	FOR z:=1 TO 100 DO
		IF  eRFID[z].nCardNumber=eLidFeederPackageState[2].nCardNumber AND eLidFeederPackageState[2].nCardNumber >0 THEN
			eRFID[z]:=eLidFeederPackageState[2];
		EXIT;
		END_IF;
	END_FOR 
			 
END_IF
END_ACTION

ACTION aP07_CapPusher:
	IF bCapPusherEnable THEN
	
	// SZLABAN **************************************************************************************************
	P07_CapPusher.IbCapPusherFormSensor;
	P07_CapPusher.bReadedCard;
	
	fbIbCapPusherFormSensor	(bIn:=	P07_CapPusher.IbCapPusherFormSensor AND 
									P07_CapPusher.bReadedCard AND
									fbPMLAuto.ePMLState = Tc3_PackML.E_PMLState.ePMLState_EXECUTE
									,tFilterTimeOn:=T#3S, tFilterTimeOff:=T#30MS);
									
	fbIbCapPusherFormSensor2	(bIn:=	P07_CapPusher.IbCapPusherFormSensor 
									,tFilterTimeOn:=T#30MS, tFilterTimeOff:=T#30MS);
	rtfbIbCapPusherFormSensor2	(CLK:=	fbIbCapPusherFormSensor2.bOUT, Q=>);
	ftbReadedCard2 				(CLK:=	P07_CapPusher.bReadedCard, Q=>);


	tonCapPusherFormNotPresent	(IN:=	iCapPusherGateCase = 20 AND 
										NOT  eCapPusherPackageState[2].bFormPresent AND
										fbIbCapPusherFormSensor.bOUT ,
									PT := T#3S); 		
										
	IF VIS_CP.bCapPusherIgnoreErrors THEN
		eCapPusherPackageState[2].bBottlePresent := TRUE;
	END_IF
	
	
	
	CASE iCapPusherGateCase OF
		
		0:
			iCapPusherGateCase		:=	iCapPusherGateCase	+	10;
		
		10: //Dojedz 2 formatka przy 1 uruchomieniu
			bCapPusherGateRun		:= FALSE;
			IF fbIbCapPusherFormSensor.bOUT THEN
				eCapPusherPackageState[2].bFormPresent		:= TRUE;
				iCapPusherGateCase							:=	iCapPusherGateCase	+	10;
			END_IF
			
		20: //Wbijanie
			IF tonCapPusherFormNotPresent.Q THEN
				itonCapPusherFormNotPresent	:=	itonCapPusherFormNotPresent + 1;
				iCapPusherGateCase			:=	iCapPusherGateCase	+	10;	
			END_IF
		
			IF (eCapPusherPackageState[2].bROPPPutted AND bFormTransportersScrewerCmdStart)  OR 
				(eCapPusherPackageState[2].bFormPresent AND NOT eCapPusherPackageState[2].bBottlePresent )
				THEN
				iCapPusherGateCase	:=	iCapPusherGateCase	+	10;	
			END_IF
			
	
		30: //Wypuszczanie 1 formatki
			bCapPusherGateRun		:= TRUE;
			IF P07_CapPusher.fbCapPusherGate.bCycleDone (*AND ftbReadedCard2.Q*) THEN
				bCapPusherGateRun						:=	FALSE;
				eCapPusherPackageState[2]				:= eClearPackageState;
				iCapPusherGateCase						:=	iCapPusherGateCase	+	10;	
			END_IF
		
		40:
			iCapPusherGateCase	:=	20;
			
	END_CASE

	ELSE
		;
	END_IF

	// KONIEC SPOWALNIACZ*********************************************************************************************
	
	
	// PODAJNIK
	IF bCapPusherEnable AND bDelayAfterStart AND NOT (P00_PackML.fbPMLAuto.ePMLState = E_PMLState.ePMLState_STOPPING)THEN
		VIS_CP.bCapPusherFeederRun := TRUE;
	ELSE
		VIS_CP.bCapPusherFeederRun := FALSE;
	END_IF
	// KONIEC PODAJNIK*************************************************************************************************
	
	
	

	// ZAKRECANIE
	
	
	eCapPusherPackageState[1].bROPPPutted;
	eCapPusherPackageState[2].bROPPPutted;;
	tonCapPusherDelay (IN:= P07_CapPusher.IbCapPusherFormSensor AND 
                   	 P07_CapPusher.bReadedCard	AND iCapPusherCase = 10 AND 
					NOT bCapPusherGateRun AND 
					bFormTransportersScrewerCmdStart
					,PT:=T#50MS);
	
	IF bCapPusherEnable AND bDelayAfterStart THEN
		
		CASE iCapPusherCase OF
			0:
				iCapPusherCase				:= iCapPusherCase	+	10;
		
			10: //Wykrywanie podjechania nowych formatek
				IF	tonCapPusherDelay.Q
 				 THEN	
					iCapPusherCase			:= iCapPusherCase	+	10;
				END_IF
				
			20:	//Rozpoczecie zakręcania
				IF NOT eCapPusherPackageState[2].bROPPPutted AND eCapPusherPackageState[2].bFormPresent AND eCapPusherPackageState[2].bBottlePresent 
				 THEN			
					VIS_CP.bCapPusherRun	:=	TRUE;
					iCapPusherCase			:= iCapPusherCase	+	10;
				END_IF
								
			30: //Czekanie na koniec zakręcania		
				IF  P07_CapPusher.fbCapPusher.bCycleDone1 THEN

					iCapPusherCase	:= iCapPusherCase	+	10;
				END_IF
			
			40: //Zapisywanie rejestrów i kasowanie sygnałów
	
				 eCapPusherPackageState[2].bROPPPutted 			:=	TRUE;
		
				FOR y:=1 TO 100 DO
					IF  eRFID[y].nCardNumber=eCapPusherPackageState[2].nCardNumber AND eCapPusherPackageState[2].nCardNumber >0 THEN
						 eRFID[y].bROPPCapped			:=	eCapPusherPackageState[2].bROPPCapped;		 
					 EXIT;
					 END_IF;
				END_FOR
		
				iCapPusherCase	:= iCapPusherCase	+	10;	 
				
			50: 
				VIS_CP.bCapPusherRun	:=	FALSE;
	
				(***Nie wykonuj dalej ruchu gdy wcisnięty stop lub błąd***)
				IF NOT (P00_PackML.fbPMLAuto.ePMLState = E_PMLState.ePMLState_STOPPING) THEN
					iCapPusherCase := 0;
				END_IF
				
		END_CASE
	ELSE
			eCapPusherPackageState[2].bROPPCapped 				:=	TRUE;

	END_IF
END_ACTION

ACTION aP07_ROPP:
IF bROPPCappingEnable THEN
	
	// SPOWALNIACZ **************************************************************************************************
	iFormBeforeROPP := 		
								BOOL_TO_INT(eBeforeROPP2PackageState[3].bFormPresent)+
								BOOL_TO_INT(eBeforeROPP2PackageState[2].bFormPresent)+
								BOOL_TO_INT(eBeforeROPP2PackageState[1].bFormPresent)+
								BOOL_TO_INT(eBeforeROPPPackageState[2].bFormPresent)+
								BOOL_TO_INT(eBeforeROPPPackageState[1].bFormPresent);
	
	
	IF bROPPSlowerEnable THEN 
	
		IF NOT fbIbROPPSevenFormSensor.bOut 
		 THEN
			bROPPSlowerCmdStart := TRUE;
		END_IF
		IF fbIbROPPSevenFormSensor.bOut 
		THEN
			bROPPSlowerCmdStart := FALSE;
		END_IF	
		IF (NOT bROPPDelayAfterStartFullRegister AND (NOT fbIbROPPThirdFormSensor.bOUT OR NOT P07_ROPP.bReadedCardBeforeROPP ))
			OR (iFormBeforeROPP<5 AND bROPPDelayAfterStartFullRegister)
		THEN
			bROPPSlowerCmdStart := TRUE;
		END_IF
	END_IF
	// KONIEC SPOWALNIACZ*********************************************************************************************
	
	// PODAJNIK
	IF bROPPFeederEnable AND bDelayAfterStart THEN
		IF iROPPCapping1Tool = 1 THEN //Praca sortera tylko dla głowicy nr 1 
			VIS_ROPP.bROPPFeederRun := TRUE;
		END_IF
	ELSE
		VIS_ROPP.bROPPFeederRun := FALSE;
	END_IF
	// KONIEC PODAJNIK*************************************************************************************************
	
	// SPRAWDZANIE NASADEK**********************************************************************************************
	IF eBeforeROPP2PackageState[3].bROPPPuttedChecked THEN
		FOR rpc1 := 1 TO 100 DO	
			 IF eBeforeROPP2PackageState[3].nCardNumber = eRFID[rpc1].nCardNumber THEN
				rpc:=rpc1;
						eRFID[rpc].bFormPresent 		:= TRUE;		
						eRFID[rpc].bROPPPutted 			:= eBeforeROPP2PackageState[3].bROPPPutted;
						eRFID[rpc].bROPPPuttedChecked 	:= eBeforeROPP2PackageState[3].bROPPPuttedChecked;	
						IF eBeforeROPP2PackageState[3].bROPPPutted THEN						
							eRFID[rpc].bBottlePresent 	:= TRUE;							
						END_IF								
						EXIT;	
			END_IF	
		END_FOR
	END_IF	
	IF eBeforeROPP2PackageState[2].bROPPPuttedChecked THEN
		FOR rpc1 := 1 TO 100 DO	
			 IF eBeforeROPP2PackageState[2].nCardNumber = eRFID[rpc1].nCardNumber THEN
				rpc:=rpc1;
						eRFID[rpc].bFormPresent 		:= TRUE;		
						eRFID[rpc].bROPPPutted 			:= eBeforeROPP2PackageState[2].bROPPPutted;
						eRFID[rpc].bROPPPuttedChecked 	:= eBeforeROPP2PackageState[2].bROPPPuttedChecked;	
						IF eBeforeROPP2PackageState[2].bROPPPutted THEN						
							eRFID[rpc].bBottlePresent 	:= TRUE;							
						END_IF								
						EXIT;	
			END_IF	
		END_FOR
	END_IF	
	IF eBeforeROPP2PackageState[1].bROPPPuttedChecked THEN
		FOR rpc1 := 1 TO 100 DO
			IF eBeforeROPP2PackageState[1].nCardNumber = eRFID[rpc1].nCardNumber THEN
				rpc:=rpc1;
					eRFID[rpc].bFormPresent 			:= TRUE;
					eRFID[rpc].bROPPPutted 				:= eBeforeROPP2PackageState[1].bROPPPutted;
					eRFID[rpc].bROPPPuttedChecked		:= eBeforeROPP2PackageState[1].bROPPPuttedChecked;	
					IF eBeforeROPP2PackageState[1].bROPPPutted THEN						
						eRFID[rpc].bBottlePresent		:= TRUE;							
					END_IF							
					EXIT;	
			END_IF	
		END_FOR
	END_IF
	// KONIEC SPRAWDZANIA NASADEK*******************************************************************************************
		
	// STOPER***************************************************************************************************************
	// w P07_ROPP	
	// KONIEC STOPER********************************************************************************************************
	
	// PRZECIAGANIE*********************************************************************************************************
	bROPPDelayAfterStartFullRegister;
	IF tonDelayAfterStart.Q AND fbIbROPPThirdFormSensor.bOUT AND tonbReadedCardBeforeROPP.Q AND NOT bROPPDelayAfterStartFullRegister AND 
		NOT  P07_ROPP.IbROPPAfter2FormSensor AND NOT fbIbROPPAfterFormSensor.bOUT 
		THEN
			eBeforeROPPCapControlPackageState[1].bFormPresent	:= TRUE;
			eBeforeROPP2PackageState[3].bFormPresent	:= TRUE;
			eBeforeROPP2PackageState[2].bFormPresent	:= TRUE;
			eBeforeROPP2PackageState[1].bFormPresent	:= TRUE;
			eBeforeROPPPackageState[2].bFormPresent		:= TRUE;
			eBeforeROPPPackageState[1].bFormPresent		:= TRUE;
			bROPPDelayAfterStartFullRegister			:= TRUE;
	END_IF
	
	IF ftIbROPPAfterFormSensor.Q THEN//Liczenie za
		iROPPAfterFormCounter :=	iROPPAfterFormCounter + 1;
	END_IF
	IF tonROPPAfterFormSensor.Q  THEN
		iROPPAfterFormCounter	:=	2;
	END_IF
	
	IF tonDelayAfterStart6s.Q  THEN 
		IF 	NOT P07_ROPP.fbROPPDrag.bCycleDone THEN
			
			IF tonROPPThirdFormSensor.Q THEN
				GVL_ROPP.bROPPDragPrepareRun					:= TRUE;
			END_IF
			
			IF	//bDragTest AND
				bROPPDelayAfterStartFullRegister AND
				(eBeforeROPPPackageState[1].bFormPresent AND eBeforeROPPPackageState[2].bFormPresent AND eBeforeROPP2PackageState[1].bFormPresent) AND
				(bROPPReady OR NOT bROPPCappingEnable) AND	
				tonROPPThirdFormSensor.Q AND tonDelayAfterStart.Q  AND iROPPAfterFormCounter >= 2 AND
				(NOT fbIbROPPAfter3FormSensor.bOUT OR NOT bROPPCappingEnable) AND (*opcja nie zatrzymywania transportera bo nadruk*)
				NOT fbROPPIbCapSorterBeforeFourthFormCheckFormSensor.bOUT AND //Jeżeli coś sie stało pod sorterem nakretek
				NOT (P00_PackML.fbPMLAuto.ePMLState = E_PMLState.ePMLState_STOPPING) 
			THEN 
				bDragTest										;//:= FALSE;
				iROPPAfterFormCounter							:= 0;
				VIS_ROPP.bROPPDragRun							:= TRUE;
			END_IF
		END_IF	
		IF P07_ROPP.fbROPPDrag.bCycleDone THEN
			VIS_ROPP.bROPPDragRun								:= FALSE;
			GVL_ROPP.bROPPDragPrepareRun						:= FALSE;
		END_IF
	END_IF
	IF P00_PackML.fbPMLAuto.ePMLState = E_PMLState.ePMLState_STOPPING THEN
		VIS_ROPP.bROPPDragRun				:= FALSE;
		GVL_ROPP.bROPPDragPrepareRun		:= FALSE;
	END_IF
	// KOENIC PRZECIAGANIE**************************************************************************************************
	
	
	// ZAKRECANIE
	eUnderROPPPackageState[1].bROPPPuttedChecked;
	eUnderROPPPackageState[1].bROPPPutted;
	eUnderROPPPackageState[1].bROPPCapped;
	eUnderROPPPackageState[1].bROPPCappingAborted;
	eUnderROPPPackageState[1].tROPPCappingTime;
	eUnderROPPPackageState[1].bROPPCappingOK;
	eUnderROPPPackageState[1].bROPPCappingChecked;
	
	tonROPPStartCappingDelay();
	tonROPPStartCappingDelay.IN:=	(P00_PackML.fbPMLAuto.ePMLState = E_PMLState.ePMLState_EXECUTE) AND
								(
								(eUnderROPPPackageState[1].bFormPresent) AND
								(NOT eUnderROPPPackageState[1].bROPPCapped AND NOT eUnderROPPPackageState[1].bROPPCappingAborted )
									
								) AND
								
								(
								(eUnderROPPPackageState[2].bFormPresent) AND 
								(NOT eUnderROPPPackageState[2].bROPPCapped AND NOT eUnderROPPPackageState[2].bROPPCappingAborted )
	
								)
	;
	tonROPPStartCappingDelay.PT:=INT_TO_TIME(300);
	
	tofbROPPCappingRunEngine	(IN:=	eUnderROPPPackageState[1].bBottlePresent OR eUnderROPPPackageState[2].bBottlePresent OR
										eBeforeROPPPackageState[1].bBottlePresent OR eBeforeROPPPackageState[2].bBottlePresent OR
										eBeforeROPP2PackageState[1].bBottlePresent OR eBeforeROPP2PackageState[2].bBottlePresent OR eBeforeROPP2PackageState[3].bBottlePresent 
								,PT:=T#10S);
	
	IF bROPPCappingEnable  THEN
		
		bROPPCappingRunEngine		:=	tofbROPPCappingRunEngine.Q;
	
		CASE iROPPCappingCase OF
			0:
				iROPPCappingCase	:= 1;
		
			1: //Wykrywanie podjechania nowych wózków i opóźnienie
				IF	tonROPPStartCappingDelay.Q  THEN	
					iROPPCappingCase	:= 2;
				END_IF
				
			2:	//Rozpoczecie zakręcania
				IF bROPPCappingEnable AND eUnderROPPPackageState[1].bBottlePresent AND eUnderROPPPackageState[1].bROPPPutted AND (eUnderROPPPackageState[1].bWeightOK OR NOT bWeight1Enable) AND eUnderROPPPackageState[1].nCardNumber > 0 
				 THEN			
					VIS_ROPP.bROPPCappingRun1 										:=	TRUE;
				END_IF
					
				IF bROPPCappingEnable AND eUnderROPPPackageState[2].bBottlePresent AND eUnderROPPPackageState[2].bROPPPutted AND (eUnderROPPPackageState[2].bWeightOK OR NOT bWeight1Enable) AND eUnderROPPPackageState[2].nCardNumber > 0 
				THEN			
					VIS_ROPP.bROPPCappingRun2 										:=	TRUE;
				END_IF
				iROPPCappingCase	:= 3;
				
			3: //Czekanie na koniec zakręcania		
				IF (
					VIS_ROPP.bROPPCappingRun1  AND (P07_ROPP.fbROPPCapping.bCycleDone1 OR P07_ROPP.fbROPPCapping.bCycleNotDone1)
					OR NOT VIS_ROPP.bROPPCappingRun1 
					) 
					AND
					(
					VIS_ROPP.bROPPCappingRun2  AND (P07_ROPP.fbROPPCapping.bCycleDone2 OR P07_ROPP.fbROPPCapping.bCycleNotDone2)
					OR NOT VIS_ROPP.bROPPCappingRun2 
					)
					THEN
						iROPPCappingCase	:= 4;
				END_IF
			
			4: //Zapisywanie rejestrów i kasowanie sygnałów
	
				eUnderROPPPackageState[1].tROPPCappingTime 				:=	P07_ROPP.fbROPPCapping.tCycleTime;
				eUnderROPPPackageState[2].tROPPCappingTime 				:=	P07_ROPP.fbROPPCapping.tCycleTime;		
				
				IF P07_ROPP.fbROPPCapping.bCycleDone1 THEN
					eUnderROPPPackageState[1].bROPPCapped 				:=	TRUE;
				ELSIF P07_ROPP.fbROPPCapping.bCycleNotDone1 THEN
					eUnderROPPPackageState[1].bROPPCapped				:=	FALSE;
					eUnderROPPPackageState[1].bROPPCappingAborted		:=	TRUE;
				ELSIF NOT bROPPCappingEnable THEN
					eUnderROPPPackageState[1].bROPPCapped				:=	TRUE;
				ELSE // Jak wyłączona
					//eUnderROPPPackageState[1].bROPPCapped				:=	TRUE; 
					eUnderROPPPackageState[1].bROPPCappingAborted		:=	TRUE;
				END_IF
	
				IF P07_ROPP.fbROPPCapping.bCycleDone2 THEN
					eUnderROPPPackageState[2].bROPPCapped 				:=	TRUE;
				ELSIF P07_ROPP.fbROPPCapping.bCycleNotDone2 THEN
					eUnderROPPPackageState[2].bROPPCapped				:=	FALSE;
					eUnderROPPPackageState[2].bROPPCappingAborted		:=	TRUE;
				ELSIF NOT bROPPCappingEnable THEN
					eUnderROPPPackageState[2].bROPPCapped				:=	TRUE;
				ELSE // Jak wyłączona
					//eUnderROPPPackageState[2].bROPPCapped				:=	TRUE; 
					eUnderROPPPackageState[2].bROPPCappingAborted		:=	TRUE;
				END_IF
							
				FOR y:=1 TO 100 DO
					IF  eRFID[y].nCardNumber=eUnderROPPPackageState[1].nCardNumber AND eUnderROPPPackageState[1].nCardNumber >0 THEN
						 //eRFID[y]:=eUnderROPPPackageState[1];
						 eRFID[y].bROPPCapped			:=	eUnderROPPPackageState[1].bROPPCapped;
						 eRFID[y].bROPPCappingAborted	:=	eUnderROPPPackageState[1].bROPPCappingAborted;				 
					 EXIT;
					 END_IF;
				END_FOR
				 
				FOR z:=1 TO 100 DO
					IF  eRFID[z].nCardNumber=eUnderROPPPackageState[2].nCardNumber AND eUnderROPPPackageState[2].nCardNumber >0 THEN
						//eRFID[z]:=eUnderROPPPackageState[2];
						 eRFID[z].bROPPCapped			:=	eUnderROPPPackageState[2].bROPPCapped;
						 eRFID[z].bROPPCappingAborted	:=	eUnderROPPPackageState[2].bROPPCappingAborted;			
					 EXIT;
					END_IF;
				END_FOR 			 	
				iROPPCappingCase := 5; 	 
			5: 
				VIS_ROPP.bROPPCappingRun1											:=	FALSE;
				VIS_ROPP.bROPPCappingRun2 											:=	FALSE;
	
				(***Nie wykonuj dalej ruchu gdy wcisnięty stop lub błąd***)
				IF NOT (P00_PackML.fbPMLAuto.ePMLState = E_PMLState.ePMLState_STOPPING) THEN
					iROPPCappingCase := 0;
				END_IF
				
		END_CASE
	ELSE
		eUnderROPPPackageState[1].bROPPCapped 				:=	TRUE;
		eUnderROPPPackageState[2].bROPPCapped 				:=	TRUE;	
		FOR y:=1 TO 100 DO
			IF  eRFID[y].nCardNumber=eUnderROPPPackageState[1].nCardNumber AND eUnderROPPPackageState[1].nCardNumber >0 THEN
				 //eRFID[y]:=eUnderROPPPackageState[1];
				 eRFID[y].bROPPCapped			:=	eUnderROPPPackageState[1].bROPPCapped;
				 eRFID[y].bROPPCappingAborted	:=	eUnderROPPPackageState[1].bROPPCappingAborted;	
			EXIT;
			END_IF;
		 END_FOR
				 
		FOR z:=1 TO 100 DO
			IF  eRFID[z].nCardNumber=eUnderROPPPackageState[2].nCardNumber AND eUnderROPPPackageState[2].nCardNumber >0 THEN
				//eRFID[z]:=eUnderROPPPackageState[2];
				eRFID[z].bROPPCapped			:=	eUnderROPPPackageState[2].bROPPCapped;
				eRFID[z].bROPPCappingAborted	:=	eUnderROPPPackageState[2].bROPPCappingAborted;	
			EXIT;
			END_IF;
		END_FOR 		 
	END_IF
	// KONIEC ZAKRECANIA
	
	
	// SPRAWDZANIE ZAKRECANIA
	eUnderROPPCorrectCapPackageState[1].bROPPCappingOK;
	eUnderROPPCorrectCapPackageState[1].bROPPCappingChecked;
	IF fbbReadedCardAfterROPP.bOUT AND eUnderROPPCorrectCapPackageState[1].bFormPresent THEN 
				
		IF VIS_ROPP.bROPPCappingCheckOK THEN				
			eUnderROPPCorrectCapPackageState[1].bROPPCappingOK			:=	TRUE;
			eUnderROPPCorrectCapPackageState[1].bBottlePresent			:=	TRUE;								
		END_IF
		eUnderROPPCorrectCapPackageState[1].bROPPCappingChecked			:=	TRUE; 		
										
		FOR rcc := 1 TO 100 DO
														
			 IF eUnderROPPCorrectCapPackageState[1].nCardNumber = eRFID[rcc].nCardNumber AND eUnderROPPCorrectCapPackageState[1].nCardNumber > 0 
			THEN		 
				rcc1:=rcc; eRFID[rcc1].bROPPCappingOK; eRFID[rcc1].bROPPCappingChecked;		                                      					
				eRFID[rcc1].bROPPCappingOK										:=	eUnderROPPCorrectCapPackageState[1].bROPPCappingOK;	
				eRFID[rcc1].bROPPCappingChecked									:=	eUnderROPPCorrectCapPackageState[1].bROPPCappingChecked	;
				IF 	eUnderROPPCorrectCapPackageState[1].bBottlePresent AND NOT eRFID[rcc].bBottlePresent THEN
					eRFID[rcc1].bBottlePresent									:=	TRUE;
					iTestBot:=iTestBot+1;
					
				END_IF				
				EXIT;
			END_IF
			
		END_FOR		
		
	END_IF
	// KONIEC SPRAWDZANIA ZAKRECANIA
	
	IF bTestBot THEN
		iTestBot:=0;
		FOR rcc := 1 TO 100 DO
			IF  eRFID[rcc].nCardNumber > 0 AND  eRFID[rcc].bFormPresent AND eRFID[rcc].bBottlePresent THEN
					iTestBot:=iTestBot+1;
			END_IF
			IF iTestBot>1 THEN
				BtESTbOT1:=true;
			END_IF
		END_FOR
	END_IF
	
ELSE
	;
END_IF
END_ACTION

ACTION aP08_CapFeeder:
IF bCapFeederEnable AND bDelayAfterStart THEN
	VIS.bCapFeederRun := TRUE;
ELSE
	VIS.bCapFeederRun := FALSE;
END_IF

IF P00_PackML.fbPMLAuto.ePMLState = E_PMLState.ePMLState_STOPPING THEN
		VIS.bCapFeederRun := FALSE;
END_IF
END_ACTION

ACTION aP08_CapSorter:
VIS.bCapSorterDragRun;
GVL.bCapSorterDragPrepareRun;

aP08_CapSorterCycleTime();

//Reset zmiennych jeśli mamy Stopping
//{warning 'CapSorter - wylaczoany Run gdy stopping'}
(*IF P00_PackML.fbPMLAuto.ePMLState = E_PMLState.ePMLState_STOPPING THEN
	GVL.bCapSorterDragPrepareRun							:= FALSE;
	VIS.bCapSorterDragRun									:= FALSE;
END_IF*)

(**** Rozpoczynanie cyklu ***)
//Dojechanie do pełna formatkami przed zakręcarką i ustawienie rejestru, dlatego że zależnie od ilości
//formatek jest różna ilość formatek przed zakręcarkami		
//Kasowanie bitu w PackML Idle	
(*bDelayAfterStartCapSorterFullRegister;
// Jeżeli formatki dojechały do końca to ustaw rejestry po 3 sekundach
IF tonCapSorterDelayAfterStart.Q AND MAIN.fbFilteredCapSorterFormsSensorGate.bOUT AND NOT bDelayAfterStartCapSorterFullRegister THEN
	eBeforeGateCapSorterPackageState[1].bFormPresent		:= TRUE;
	//eBeforeCapSorterPackageState[4].bFormPresent			:= TRUE;
	//eBeforeCapSorterPackageState[3].bFormPresent			:= TRUE;
	//eBeforeCapSorterPackageState[2].bFormPresent			:= TRUE;
	//eBeforeCapSorterPackageState[1].bFormPresent			:= TRUE;
	bDelayAfterStartCapSorterFullRegister					:= TRUE;
	ibDelayAfterStartCapSorterFullRegister	:=	ibDelayAfterStartCapSorterFullRegister	+	1;
END_IF //dp*)


(*** ROZPOCZECIE KONFEKCJI PO RESECIE CYKLU***)
// Wykonanie jednego przeciągania, żeby pozbyć się formatek do 0
// po 1 uruchomieniu po 60sek
(*tonLongDelayAfterStart.ET;tonLongDelayAfterStart.Q;
IF (P00_PackML.rttonLongDelayAfterStart.Q OR brtCapSorterLongDelayFirstDraging) AND tonIbCapSorterAfterFormSensor.Q  AND tonIbCapSorterFirstFormCheckFormSensor.Q  THEN
	brtCapSorterLongDelayFirstDraging							:= TRUE;
	//IF tonCapSorterFourthFormatSensor.Q THEN //Przeciagaj jak 3
		brtCapSorterLongDelayFirstDraging						:= FALSE;
		VIS.bCapSorterDragRun									:= TRUE; 
	//END_IF
	IF P08_CapSorter.fbCapSorterDragStation.bCycleDone THEN
		VIS.bCapSorterDragRun									:= FALSE;
		GVL.bCapSorterDragPrepareRun							:= FALSE;
		brtCapSorterLongDelayFirstDraging						:= FALSE;			
	END_IF
END_IF*)

//bCapSorterDragIfNot4PucksAnd5s
tonCapSorterDragIfNot4PucksAnd5s	(IN:=
		P00_PackML.fbPMLAuto.ePMLState = E_PMLState.ePMLState_EXECUTE AND
		(P08_CapSorter.fbCapSorterDragStation.eState = E_Station.eReady OR P08_CapSorter.fbCapSorterDragStation.eRunningState = E_DragStationState.eLifting) AND	
		tonIbCapSorterFirstFormCheckFormSensor.Q AND NOT stCapSorterRead.eReservedSignals.bReserved00 AND
		NOT fbIbCapSorterFourthFormCheckFormSensor.bOut AND
		NOT MAIN.IbCapSorterBeforeFourthFormCheckFormSensor AND
		tonIbCapSorterAfterFormSensor.Q AND NOT tonIbCapSorterAfterFormSensor3.Q AND
		tonDelayAfterStart.Q
		, PT:=T#1S000MS);	
IF (tonCapSorterDragIfNot4PucksAnd5s.Q OR bCapSorterDragIfNot4PucksAnd5s) THEN
		bCapSorterDragIfNot4PucksAnd5s							:= TRUE;
		VIS.bCapSorterDragRun									:= TRUE; 
	IF P08_CapSorter.fbCapSorterDragStation.bCycleDone THEN
		VIS.bCapSorterDragRun									:= FALSE;
		GVL.bCapSorterDragPrepareRun							:= FALSE;
		bCapSorterDragIfNot4PucksAnd5s							:= FALSE;	
		eBeforeGateCapSorterPackageState[1].bFormPresent		:= FALSE;
		eBeforeCapSorterPackageState[4].bFormPresent			:= FALSE;
		eBeforeCapSorterPackageState[3].bFormPresent			:= FALSE;
		eBeforeCapSorterPackageState[2].bFormPresent			:= FALSE;
		eBeforeCapSorterPackageState[1].bFormPresent			:= FALSE;
	END_IF
END_IF
//Koniec bCapSorterDragIfNot4PucksAnd5s

//Licz. form.
tonCapSorterDragFormCounter4	(IN:=iCapSorterDragFormCounter <> 4 AND fbIbCapSorterFourthFormCheckFormSensor.bOut, PT:=T#10S);//bylo 50
tonCapSorterDragFormCounter4b	(IN:=iCapSorterDragFormCounter > 4 AND fbIbCapSorterFourthFormCheckFormSensor.bOut AND bFormTransportersScrewerCmdStart, PT:=T#10S); //Na testy
tonCapSorterDragFormCounter4.ET;
IF tonCapSorterDragFormCounter4.Q THEN
	iCapSorterDragFormCounter := 4;
	itonCapSorterDragFormCounter4	:=	itonCapSorterDragFormCounter4	+	1;
END_IF
IF tonCapSorterDragFormCounter4b.Q THEN
	iCapSorterDragFormCounter := 4;
	itonCapSorterDragFormCounter4b	:=	itonCapSorterDragFormCounter4b	+	1;	
END_IF

IF 	P08_CapSorter.fbCapSorterDragStation.eRunningState = E_DragStationState.eDraging THEN
	iCapSorterDragFormCounter				:= 0;
END_IF

IF 	P08_CapSorter.fbCapSorterDragStation.eRunningState = E_DragStationState.eEndingOfDrag 
	OR (bFormTransportersScrewerStop AND fbTransporterQueues.bOUT) // Blokada kolejek do testów
THEN
	bFormTransportersScrewerStop			:= FALSE;
END_IF


IF tonDelayAfterStart6s.Q AND NOT brtCapSorterLongDelayFirstDraging AND NOT bCapSorterDragIfNot4PucksAnd5s THEN 

	   	//4 Formatka stoi na czujniku prze czas T
		IF	
			//tonCapSorterFourthFormatSensorAnRegister.Q AND 
			//fbIbCapSorterFourthFormCheckFormSensor.bOUT AND
			tonIbCapSorterFirstFormCheckFormSensor.Q AND
			NOT (P00_PackML.fbPMLAuto.ePMLState = E_PMLState.ePMLState_STOPPING) 
		THEN
			GVL.bCapSorterDragPrepareRun						:= TRUE;
		END_IF


	IF 
		eBeforeCapSorterPackageState[1].bFormPresent AND eBeforeCapSorterPackageState[2].bFormPresent AND 
	   	eBeforeCapSorterPackageState[3].bFormPresent AND eBeforeCapSorterPackageState[4].bFormPresent AND 
		NOT P08_CapSorter.fbCapSorterDragStation.bCycleDone THEN
		
	   	//4 Formatka stoi na czujniku prze czas T
		(*IF	
			tonCapSorterFourthFormatSensorAnRegister.Q AND 
			NOT (P00_PackML.fbPMLAuto.ePMLState = E_PMLState.ePMLState_STOPPING) 
		THEN
			GVL.bCapSorterDragPrepareRun						:= TRUE;
		END_IF*)
	
		//Wykonały cykl lub nie było butelki
		IF ((eCapSorterPackageState[1].bFormPresent AND eCapSorterPackageState[1].bBottlePresent AND (eCapSorterPackageState[1].bCapSorterPutted OR  eCapSorterPackageState[1].bCapSorterPuttedAborted) OR (NOT eCapSorterPackageState[1].bWeightOK AND bCapSorterOnlyWeightOKEnable) OR (NOT eCapSorterPackageState[1].bROPPCapped AND bROPPCappingEnable)) OR NOT eCapSorterPackageState[1].bBottlePresent OR NOT eCapSorterPackageState[1].bFormPresent) AND
		   ((eCapSorterPackageState[2].bFormPresent AND eCapSorterPackageState[2].bBottlePresent AND (eCapSorterPackageState[2].bCapSorterPutted OR  eCapSorterPackageState[2].bCapSorterPuttedAborted) OR (NOT eCapSorterPackageState[2].bWeightOK AND bCapSorterOnlyWeightOKEnable) OR (NOT eCapSorterPackageState[2].bROPPCapped AND bROPPCappingEnable)) OR NOT eCapSorterPackageState[2].bBottlePresent OR NOT eCapSorterPackageState[2].bFormPresent) AND
		   ((eCapSorterPackageState[3].bFormPresent AND eCapSorterPackageState[3].bBottlePresent AND (eCapSorterPackageState[3].bCapSorterPutted OR  eCapSorterPackageState[3].bCapSorterPuttedAborted) OR (NOT eCapSorterPackageState[3].bWeightOK AND bCapSorterOnlyWeightOKEnable) OR (NOT eCapSorterPackageState[3].bROPPCapped AND bROPPCappingEnable)) OR NOT eCapSorterPackageState[3].bBottlePresent OR NOT eCapSorterPackageState[3].bFormPresent) AND
		   ((eCapSorterPackageState[4].bFormPresent AND eCapSorterPackageState[4].bBottlePresent AND (eCapSorterPackageState[4].bCapSorterPutted OR  eCapSorterPackageState[4].bCapSorterPuttedAborted) OR (NOT eCapSorterPackageState[4].bWeightOK AND bCapSorterOnlyWeightOKEnable) OR (NOT eCapSorterPackageState[4].bROPPCapped AND bROPPCappingEnable)) OR NOT eCapSorterPackageState[4].bBottlePresent OR NOT eCapSorterPackageState[4].bFormPresent) THEN
		
		   	//Rejest za pusty i możemy przeciągać
			IF NOT 	eAfterCapSorterPackageState[1].bFormPresent AND NOT eAfterCapSorterPackageState[2].bFormPresent AND NOT eAfterCapSorterPackageState[3].bFormPresent AND NOT eAfterCapSorterPackageState[4].bFormPresent AND
				 	tonIbCapSorterAfterFormSensor.Q AND NOT tonIbCapSorterAfterFormSensor3.Q AND
					(
				 	(tonCapSorterFourthFormatSensorAnRegister.Q AND		iCapSorterDragFormCounter = 4 AND tonLongDelayAfterStart.Q) OR 
					(tonCapSorterFourthFormatSensorStarting.Q	AND NOT tonLongDelayAfterStart.Q) // przy 1 uruch
					)
					AND 
					tonIbCapSorterFirstFormCheckFormSensor.Q AND NOT stCapSorterRead.eReservedSignals.bReserved00 AND
					(NOT stCapSorterRead.bEnable OR NOT bCapSorterRobotPlaceDone OR bCapSorterDisable)  AND
					{warning 'MANTZ -CapSorter - wylaczoany PlaceDone'}
					//(NOT stCapSorterRead.bEnable  OR bCapSorterDisable) 
					//AND NOT fbIbBlowBeforeGripperScrewerSensor2.bOUT
					tonbFormTransportersAfterCapSorterCmdStart.Q
					AND NOT (P00_PackML.fbPMLAuto.ePMLState = E_PMLState.ePMLState_STOPPING) 					
				THEN
					VIS.bCapSorterDragRun					:= TRUE;
					bCapSorterRobotPreparePlace				:= FALSE; // Nowe
					bCapSorterBeforeRobotBottleAndNoCap1	:= FALSE; // Nowe
					bCapSorterBeforeRobotBottleAndNoCap2	:= FALSE; // Nowe
					bCapSorterBeforeRobotBottleAndNoCap3	:= FALSE; // Nowe
					bCapSorterBeforeRobotBottleAndNoCap4	:= FALSE; // Nowe	
					
					(*Opcją z transporterem ROPP i wyewaniem*)				
					IF MAIN.IbCapSorterBeforeFourthFormCheckFormSensor AND NOT bROPPCappingEnable THEN
						bCapSorterDragIfNot4PucksAnd5sRepair	:= TRUE;
					END_IF
			END_IF 
		END_IF  
	END_IF	
	
	//CycleDone, resetuje pozwolenia
	IF P08_CapSorter.fbCapSorterDragStation.bCycleDone THEN
		VIS.bCapSorterDragRun								:= FALSE;
		GVL.bCapSorterDragPrepareRun						:= FALSE;
	END_IF
	tonStoppingCapSorter(IN:=(P00_PackML.fbPMLAuto.ePMLState = E_PMLState.ePMLState_STOPPING) AND P08_CapSorter.fbCapSorterDragStation.eRunningState = E_DragStationState.eLifting, PT:=T#0S); //bylo 10s
	IF tonStoppingCapSorter.Q  THEN //Nowe do testów
		GVL.bCapSorterDragPrepareRun						:= FALSE;
	END_IF
	
END_IF

(************************************************************************************)
//Deklaracja opóźnienia startu nakladania
tonCapSorterDelay(	IN:=	P00_PackML.fbPMLAuto.ePMLState = E_PMLState.ePMLState_EXECUTE AND
							eCapSorterPackageState[1].bFormPresent OR //AND 
							eCapSorterPackageState[2].bFormPresent OR //AND 
							eCapSorterPackageState[3].bFormPresent OR //AND 
							eCapSorterPackageState[4].bFormPresent 
					,PT:=INT_TO_TIME(300));

tonCapSorterDelay2(	IN:= iCapSorterCase = 3 AND 
						(stCapSorterRead.ePackMLAutoState = E_PMLState.ePMLState_EXECUTE OR stCapSorterRead.ePackMLAutoState = E_PMLState.ePMLState_STOPPING) AND 
						NOT (P00_PackML.fbPMLAuto.ePMLState = E_PMLState.ePMLState_STOPPING) 
					,PT:=T#700MS);

IF stCapSorterRead.bEnable AND NOT bCapSorterDisable AND NOT bChangeOver THEN
	
	IF iCapSorterCase > 4  AND NOT VIS.bCapSorterDragRun THEN//NOT Run bo miały się kasować razem z przeciąganiem
		//bCapSorterRobotPreparePlace				:=	eBeforeCapSorterPackageState[1].bFormPresent	AND eBeforeCapSorterPackageState[2].bFormPresent AND eBeforeCapSorterPackageState[3].bFormPresent AND eBeforeCapSorterPackageState[4].bFormPresent;
		IF eBeforeCapSorterPackageState[1].bFormPresent	AND eBeforeCapSorterPackageState[2].bFormPresent AND eBeforeCapSorterPackageState[3].bFormPresent AND eBeforeCapSorterPackageState[4].bFormPresent THEN
			bCapSorterRobotPreparePlace				:=	bCapSorterBeforeRobotBottleAndNoCap1 OR bCapSorterBeforeRobotBottleAndNoCap2 OR 
														bCapSorterBeforeRobotBottleAndNoCap3 OR bCapSorterBeforeRobotBottleAndNoCap4;																				
			bCapSorterBeforeRobotBottleAndNoCap1	:=	eBeforeCapSorterPackageState[1].bFormPresent AND eBeforeCapSorterPackageState[1].bBottlePresent AND (eBeforeCapSorterPackageState[1].bWeightOK OR NOT bCapSorterOnlyWeightOKEnable) AND (eBeforeCapSorterPackageState[1].bROPPCapped OR NOT bROPPCappingEnable);
			bCapSorterBeforeRobotBottleAndNoCap2	:=	eBeforeCapSorterPackageState[2].bFormPresent AND eBeforeCapSorterPackageState[2].bBottlePresent AND (eBeforeCapSorterPackageState[2].bWeightOK OR NOT bCapSorterOnlyWeightOKEnable) AND (eBeforeCapSorterPackageState[2].bROPPCapped OR NOT bROPPCappingEnable);
			bCapSorterBeforeRobotBottleAndNoCap3	:=	eBeforeCapSorterPackageState[3].bFormPresent AND eBeforeCapSorterPackageState[3].bBottlePresent AND (eBeforeCapSorterPackageState[3].bWeightOK OR NOT bCapSorterOnlyWeightOKEnable) AND (eBeforeCapSorterPackageState[3].bROPPCapped OR NOT bROPPCappingEnable);
			bCapSorterBeforeRobotBottleAndNoCap4	:=	eBeforeCapSorterPackageState[4].bFormPresent AND eBeforeCapSorterPackageState[4].bBottlePresent AND (eBeforeCapSorterPackageState[4].bWeightOK OR NOT bCapSorterOnlyWeightOKEnable) AND (eBeforeCapSorterPackageState[4].bROPPCapped OR NOT bROPPCappingEnable);
		END_IF
	END_IF	

	CASE iCapSorterCase OF
		0:
			(***Nie wykonuj dalej ruchu gdy wcisnięty stop lub błąd***)
			IF NOT (P00_PackML.fbPMLAuto.ePMLState = E_PMLState.ePMLState_STOPPING) THEN
				iCapSorterCase	:= 1;
			END_IF
			
		1: //Wykrywanie 
			IF	tonCapSorterDelay.Q  THEN	
				iCapSorterCase	:= 2;
			END_IF
			
		2:	//Przygotowani			
			
			bCapSorterRobotPlace; 
			bCapSorterRobotBottleAndNoCap1			:= eCapSorterPackageState[1].bFormPresent AND eCapSorterPackageState[1].bBottlePresent AND (NOT eCapSorterPackageState[1].bCapSorterPutted) AND NOT (eCapSorterPackageState[1].bCapSorterPuttedAborted)  AND (eCapSorterPackageState[1].bWeightOK OR NOT bCapSorterOnlyWeightOKEnable) AND (eCapSorterPackageState[1].bROPPCapped OR NOT bROPPCappingEnable);
			bCapSorterRobotBottleAndNoCap2			:= eCapSorterPackageState[2].bFormPresent AND eCapSorterPackageState[2].bBottlePresent AND (NOT eCapSorterPackageState[2].bCapSorterPutted) AND NOT (eCapSorterPackageState[2].bCapSorterPuttedAborted)  AND (eCapSorterPackageState[2].bWeightOK OR NOT bCapSorterOnlyWeightOKEnable) AND (eCapSorterPackageState[2].bROPPCapped OR NOT bROPPCappingEnable);
			bCapSorterRobotBottleAndNoCap3			:= eCapSorterPackageState[3].bFormPresent AND eCapSorterPackageState[3].bBottlePresent AND (NOT eCapSorterPackageState[3].bCapSorterPutted) AND NOT (eCapSorterPackageState[3].bCapSorterPuttedAborted)  AND (eCapSorterPackageState[3].bWeightOK OR NOT bCapSorterOnlyWeightOKEnable) AND (eCapSorterPackageState[3].bROPPCapped OR NOT bROPPCappingEnable);
			bCapSorterRobotBottleAndNoCap4			:= eCapSorterPackageState[4].bFormPresent AND eCapSorterPackageState[4].bBottlePresent AND (NOT eCapSorterPackageState[4].bCapSorterPutted) AND NOT (eCapSorterPackageState[4].bCapSorterPuttedAborted)  AND (eCapSorterPackageState[4].bWeightOK OR NOT bCapSorterOnlyWeightOKEnable) AND (eCapSorterPackageState[4].bROPPCapped OR NOT bROPPCappingEnable);

			//PreparePlace
			IF  
				eCapSorterPackageState[1].bFormPresent AND (NOT eCapSorterPackageState[1].bBottlePresent OR eCapSorterPackageState[1].bCapSorterPutted OR eCapSorterPackageState[1].bCapSorterPuttedAborted OR NOT eCapSorterPackageState[1].bFormPresent) AND 
				eCapSorterPackageState[2].bFormPresent AND (NOT eCapSorterPackageState[2].bBottlePresent OR eCapSorterPackageState[2].bCapSorterPutted OR eCapSorterPackageState[2].bCapSorterPuttedAborted OR NOT eCapSorterPackageState[2].bFormPresent) AND 
				eCapSorterPackageState[3].bFormPresent AND (NOT eCapSorterPackageState[3].bBottlePresent OR eCapSorterPackageState[3].bCapSorterPutted OR eCapSorterPackageState[3].bCapSorterPuttedAborted OR NOT eCapSorterPackageState[3].bFormPresent) AND  
				eCapSorterPackageState[4].bFormPresent AND (NOT eCapSorterPackageState[4].bBottlePresent OR eCapSorterPackageState[4].bCapSorterPutted OR eCapSorterPackageState[4].bCapSorterPuttedAborted OR NOT eCapSorterPackageState[4].bFormPresent)

			 THEN
				//bCapSorterRobotPreparePlace			:= eBeforeCapSorterPackageState[1].bFormPresent	AND eBeforeCapSorterPackageState[2].bFormPresent AND eBeforeCapSorterPackageState[3].bFormPresent AND eBeforeCapSorterPackageState[4].bFormPresent;			
				IF eBeforeCapSorterPackageState[1].bFormPresent	AND eBeforeCapSorterPackageState[2].bFormPresent AND eBeforeCapSorterPackageState[3].bFormPresent AND eBeforeCapSorterPackageState[4].bFormPresent //THEN
					AND NOT VIS.bCapSorterDragRun THEN//NOT Run bo miały się kasować razem z przeciąganiem
	
					bCapSorterRobotPreparePlace				:=	bCapSorterBeforeRobotBottleAndNoCap1 OR bCapSorterBeforeRobotBottleAndNoCap2 OR 
																bCapSorterBeforeRobotBottleAndNoCap3 OR bCapSorterBeforeRobotBottleAndNoCap4;
					bCapSorterBeforeRobotBottleAndNoCap1	:= eBeforeCapSorterPackageState[1].bFormPresent AND eBeforeCapSorterPackageState[1].bBottlePresent AND (eBeforeCapSorterPackageState[1].bWeightOK OR NOT bCapSorterOnlyWeightOKEnable) AND (eBeforeCapSorterPackageState[1].bROPPCapped OR NOT bROPPCappingEnable);
					bCapSorterBeforeRobotBottleAndNoCap2	:= eBeforeCapSorterPackageState[2].bFormPresent AND eBeforeCapSorterPackageState[2].bBottlePresent AND (eBeforeCapSorterPackageState[2].bWeightOK OR NOT bCapSorterOnlyWeightOKEnable) AND (eBeforeCapSorterPackageState[2].bROPPCapped OR NOT bROPPCappingEnable);
					bCapSorterBeforeRobotBottleAndNoCap3	:= eBeforeCapSorterPackageState[3].bFormPresent AND eBeforeCapSorterPackageState[3].bBottlePresent AND (eBeforeCapSorterPackageState[3].bWeightOK OR NOT bCapSorterOnlyWeightOKEnable) AND (eBeforeCapSorterPackageState[3].bROPPCapped OR NOT bROPPCappingEnable);
					bCapSorterBeforeRobotBottleAndNoCap4	:= eBeforeCapSorterPackageState[4].bFormPresent AND eBeforeCapSorterPackageState[4].bBottlePresent AND (eBeforeCapSorterPackageState[4].bWeightOK OR NOT bCapSorterOnlyWeightOKEnable) AND (eBeforeCapSorterPackageState[4].bROPPCapped OR NOT bROPPCappingEnable);
				END_IF
			END_IF
			
			IF bCapSorterRobotBottleAndNoCap1 OR bCapSorterRobotBottleAndNoCap2 OR bCapSorterRobotBottleAndNoCap3 OR bCapSorterRobotBottleAndNoCap4 THEN
				iCapSorterCase	:= 3;
			END_IF
			
		3: //Rozpoczecie	
			IF NOT (P00_PackML.fbPMLAuto.ePMLState = E_PMLState.ePMLState_STOPPING) THEN
				IF  tonCapSorterDelay2.Q THEN
					bCapSorterRobotPlace					:=	TRUE;
					//Tutaj bo czasami zostawało w 3
					bCapSorterRobotBottleAndNoCap1			:= eCapSorterPackageState[1].bFormPresent AND eCapSorterPackageState[1].bBottlePresent AND (NOT eCapSorterPackageState[1].bCapSorterPutted) AND NOT (eCapSorterPackageState[1].bCapSorterPuttedAborted) AND (eCapSorterPackageState[1].bWeightOK OR NOT bCapSorterOnlyWeightOKEnable) AND (eCapSorterPackageState[1].bROPPCapped OR NOT bROPPCappingEnable); 
					bCapSorterRobotBottleAndNoCap2			:= eCapSorterPackageState[2].bFormPresent AND eCapSorterPackageState[2].bBottlePresent AND (NOT eCapSorterPackageState[2].bCapSorterPutted) AND NOT (eCapSorterPackageState[2].bCapSorterPuttedAborted) AND (eCapSorterPackageState[2].bWeightOK OR NOT bCapSorterOnlyWeightOKEnable) AND (eCapSorterPackageState[2].bROPPCapped OR NOT bROPPCappingEnable);  
					bCapSorterRobotBottleAndNoCap3			:= eCapSorterPackageState[3].bFormPresent AND eCapSorterPackageState[3].bBottlePresent AND (NOT eCapSorterPackageState[3].bCapSorterPutted) AND NOT (eCapSorterPackageState[3].bCapSorterPuttedAborted) AND (eCapSorterPackageState[3].bWeightOK OR NOT bCapSorterOnlyWeightOKEnable) AND (eCapSorterPackageState[3].bROPPCapped OR NOT bROPPCappingEnable);  
					bCapSorterRobotBottleAndNoCap4			:= eCapSorterPackageState[4].bFormPresent AND eCapSorterPackageState[4].bBottlePresent AND (NOT eCapSorterPackageState[4].bCapSorterPutted) AND NOT (eCapSorterPackageState[4].bCapSorterPuttedAborted) AND (eCapSorterPackageState[4].bWeightOK OR NOT bCapSorterOnlyWeightOKEnable) AND (eCapSorterPackageState[4].bROPPCapped OR NOT bROPPCappingEnable);  
					iCapSorterCase				:=	4;
				END_IF
			END_IF
		4:
			
			bCapSorterRobotPlaceAck		;
			bCapSorterRobotPlaceDone 	;
			bCapSorterRobotForm1CapPutted;
			bCapSorterRobotForm2CapPutted;
			bCapSorterRobotForm3CapPutted;
			bCapSorterRobotForm4CapPutted;
			
			//Warunek przejścia dalej, albo wykonano zakręcanie albo nie było rozkazu zakręcania (np. brak butelki)
			//IF	bCapSorterRobotPlaceDoneOR
			IF	(bCapSorterRobotPlaceAck AND bCapSorterRobotPlaceDone)	OR				
				stCapSorterRead.ePackMLAutoState = E_PMLState.ePMLState_RESETTING OR  NOT bCapSorterRobotPlace
				THEN
					iCapSorterCase	:= 5;
			END_IF
		
		5: //Zapisywanie rejestrów i kasowanie sygnałów

			eCapSorterPackageState[1].tCapSorterPuttingTime;
			eCapSorterPackageState[2].tCapSorterPuttingTime;		
			eCapSorterPackageState[3].tCapSorterPuttingTime;
			eCapSorterPackageState[4].tCapSorterPuttingTime;			
			
			IF bCapSorterRobotForm1CapPutted AND bCapSorterRobotPlaceDone THEN
				eCapSorterPackageState[1].bCapSorterPutted 				:=	TRUE;
			ELSIF bCapSorterRobotPlaceAck THEN 
				eCapSorterPackageState[1].bCapSorterPutted				:=	TRUE; 
				eCapSorterPackageState[1].bCapSorterPuttedAborted		:=	TRUE;
			END_IF
			IF bCapSorterRobotForm2CapPutted AND bCapSorterRobotPlaceDone THEN
				eCapSorterPackageState[2].bCapSorterPutted 				:=	TRUE;
			ELSIF bCapSorterRobotPlaceAck THEN 
				eCapSorterPackageState[2].bCapSorterPutted				:=	TRUE; 
				eCapSorterPackageState[2].bCapSorterPuttedAborted		:=	TRUE;
			END_IF			
			IF bCapSorterRobotForm3CapPutted AND bCapSorterRobotPlaceDone THEN
				eCapSorterPackageState[3].bCapSorterPutted 				:=	TRUE;
			ELSIF bCapSorterRobotPlaceAck THEN 
				eCapSorterPackageState[3].bCapSorterPutted				:=	TRUE; 
				eCapSorterPackageState[3].bCapSorterPuttedAborted		:=	TRUE;
			END_IF
			IF bCapSorterRobotForm4CapPutted AND bCapSorterRobotPlaceDone THEN
				eCapSorterPackageState[4].bCapSorterPutted 				:=	TRUE;
			ELSIF bCapSorterRobotPlaceAck THEN 
				eCapSorterPackageState[4].bCapSorterPutted				:=	TRUE; 
				eCapSorterPackageState[4].bCapSorterPuttedAborted		:=	TRUE;
			END_IF
			
			FOR y:=1 TO 100 DO
				IF  eRFID[y].nCardNumber=eCapSorterPackageState[1].nCardNumber AND eCapSorterPackageState[1].nCardNumber >0 THEN
					 eRFID[y]:=eCapSorterPackageState[1];
				EXIT;
				END_IF;
			 END_FOR
			
			FOR y:=1 TO 100 DO
				IF  eRFID[y].nCardNumber=eCapSorterPackageState[2].nCardNumber AND eCapSorterPackageState[2].nCardNumber >0 THEN
					 eRFID[y]:=eCapSorterPackageState[2];
				EXIT;
				END_IF;
			 END_FOR
					 
			FOR z:=1 TO 100 DO
				IF  eRFID[z].nCardNumber=eCapSorterPackageState[3].nCardNumber AND eCapSorterPackageState[3].nCardNumber >0 THEN
					eRFID[z]:=eCapSorterPackageState[3];
				EXIT;
				END_IF;
			END_FOR 
			
			FOR z:=1 TO 100 DO
				IF  eRFID[z].nCardNumber=eCapSorterPackageState[4].nCardNumber AND eCapSorterPackageState[4].nCardNumber >0 THEN
					eRFID[z]:=eCapSorterPackageState[4];
				EXIT;
				END_IF;
			END_FOR 	
			 	
			 iCapSorterCase := 6; 
			 
		6: 
			bCapSorterRobotPlace          											:=	FALSE;	
			bCapSorterRobotBottleAndNoCap1											:=	FALSE;
			bCapSorterRobotBottleAndNoCap2											:=	FALSE;
			bCapSorterRobotBottleAndNoCap3											:=	FALSE;
			bCapSorterRobotBottleAndNoCap4											:=	FALSE;
			bCapSorterRobotPreparePlace												:=	FALSE;	
			bCapSorterBeforeRobotBottleAndNoCap1									:=	FALSE;	
			bCapSorterBeforeRobotBottleAndNoCap2									:=	FALSE;	
			bCapSorterBeforeRobotBottleAndNoCap3									:=	FALSE;	
			bCapSorterBeforeRobotBottleAndNoCap4									:=	FALSE;				
			
			iCapSorterCase := 0;

	END_CASE
	
ELSE

	IF tCapSorterCycleTestTime < T#1MS THEN
		tCapSorterCycleTestTime := T#4000MS;
	END_IF
	tonCapSorterPackageState1bCapSorterPutted	(IN:= eCapSorterPackageState[1].bBottlePresent AND NOT eCapSorterPackageState[1].bCapSorterPutted, 	PT:= tCapSorterCycleTestTime);
	IF bCapSorterCycleTest THEN
		IF tonCapSorterPackageState1bCapSorterPutted.Q THEN
			eCapSorterPackageState[1].bCapSorterPutted			:=	TRUE;
			tCapSorterCycleTestTime := DINT_TO_TIME(diRandom);
		END_IF
		eCapSorterPackageState[2].bCapSorterPutted 				:=	TRUE;	
		eCapSorterPackageState[3].bCapSorterPutted 				:=	TRUE;	
		eCapSorterPackageState[4].bCapSorterPutted 				:=	TRUE;		
		
		IF 
			eBeforeCapSorterPackageState[1].bFormPresent AND
			eBeforeCapSorterPackageState[2].bFormPresent AND
			eBeforeCapSorterPackageState[3].bFormPresent AND
			eBeforeCapSorterPackageState[4].bFormPresent
		THEN
			eBeforeCapSorterPackageState[1].bBottlePresent		:= TRUE;
		END_IF
	ELSE
		eCapSorterPackageState[1].bCapSorterPutted				:=	TRUE;
		eCapSorterPackageState[2].bCapSorterPutted 				:=	TRUE;	
		eCapSorterPackageState[3].bCapSorterPutted 				:=	TRUE;	
		eCapSorterPackageState[4].bCapSorterPutted 				:=	TRUE;
	END_IF
	
	FOR y:=1 TO 100 DO
		IF  eRFID[y].nCardNumber=eCapSorterPackageState[1].nCardNumber AND eCapSorterPackageState[1].nCardNumber >0 THEN
			 eRFID[y]:=eCapSorterPackageState[1];		EXIT;		END_IF;
	 END_FOR
	
	FOR y:=1 TO 100 DO
		IF  eRFID[y].nCardNumber=eCapSorterPackageState[2].nCardNumber AND eCapSorterPackageState[2].nCardNumber >0 THEN
			 eRFID[y]:=eCapSorterPackageState[2];		EXIT;		END_IF;
	 END_FOR
			 
	FOR z:=1 TO 100 DO
		IF  eRFID[z].nCardNumber=eCapSorterPackageState[3].nCardNumber AND eCapSorterPackageState[3].nCardNumber >0 THEN
			eRFID[z]:=eCapSorterPackageState[3];		EXIT;		END_IF;
	END_FOR 
	
	FOR z:=1 TO 100 DO
		IF  eRFID[z].nCardNumber=eCapSorterPackageState[4].nCardNumber AND eCapSorterPackageState[4].nCardNumber >0 THEN
			eRFID[z]:=eCapSorterPackageState[4];		EXIT;		END_IF;
	END_FOR 	
				 
END_IF
END_ACTION

ACTION aP08_CapSorterCycleTime:

///////// TEST SYMULACJI CZASU CYKLU SORTERA
// Randomowa liczba
fbDrand(Seed:=1, Num=> );
diRandom := F_Scaling
(
rValue	:=	LREAL_TO_DINT(fbDrand.Num*1000),
rXmin	:= 0,
rXmax	:= 1000,
rYmin	:= 4000,
rYmax	:= 6000,
);


	bCapSorterCycleTest;
	tonCapSorterCycleTime.ET; 
	tonCapSorterCycleTime (IN:=
		(	// sa jakies butelki
		(eCapSorterPackageState[1].bFormPresent AND eCapSorterPackageState[1].bBottlePresent AND NOT eCapSorterPackageState[1].bCapSorterPutted AND NOT eCapSorterPackageState[1].bCapSorterPuttedAborted) OR
		(eCapSorterPackageState[2].bFormPresent AND eCapSorterPackageState[2].bBottlePresent AND NOT eCapSorterPackageState[2].bCapSorterPutted AND NOT eCapSorterPackageState[2].bCapSorterPuttedAborted) OR 
		(eCapSorterPackageState[3].bFormPresent AND eCapSorterPackageState[3].bBottlePresent AND NOT eCapSorterPackageState[3].bCapSorterPutted AND NOT eCapSorterPackageState[3].bCapSorterPuttedAborted) OR  
		(eCapSorterPackageState[4].bFormPresent AND eCapSorterPackageState[4].bBottlePresent AND NOT eCapSorterPackageState[4].bCapSorterPutted AND NOT eCapSorterPackageState[4].bCapSorterPuttedAborted)
		)	// nie ma
		OR 
		(
		eCapSorterPackageState[1].bFormPresent AND NOT eCapSorterPackageState[1].bBottlePresent	AND 
		eCapSorterPackageState[2].bFormPresent AND NOT eCapSorterPackageState[2].bBottlePresent	AND 
		eCapSorterPackageState[3].bFormPresent AND NOT eCapSorterPackageState[3].bBottlePresent	AND  
		eCapSorterPackageState[4].bFormPresent AND NOT eCapSorterPackageState[4].bBottlePresent	 AND
		(NOT eBeforeCapSorterPackageState[4].bFormPresent OR
		NOT tonIbCapSorterAfterFormSensor.Q)
		)
		
		,PT:= T#100M);
		
	fttonCapSorterCycleTime	(CLK:=tonCapSorterCycleTime.IN, Q=>);
	
	IF ics<=0 THEN ics:=1;	END_IF
	IF fttonCapSorterCycleTime.Q THEN
		AtCapSorterCycleTime[ics]	:=	ttonCapSorterCycleTimeET;
		ics							:=	ics+1;
	END_IF
	ttonCapSorterCycleTimeET := tonCapSorterCycleTime.ET;
	IF ics>=10 THEN
		FOR i:=1 TO 10 DO
			AtCapSorterCycleTime[i]	:=	T#0S;
		END_FOR
		ics := 1;
	END_IF
		AtCapSorterCycleTime[1];
		AtCapSorterCycleTime[2];
		AtCapSorterCycleTime[3];
		AtCapSorterCycleTime[4];
		AtCapSorterCycleTime[5];
		AtCapSorterCycleTime[6];
		AtCapSorterCycleTime[7];
		AtCapSorterCycleTime[8];
		AtCapSorterCycleTime[9];
		AtCapSorterCycleTime[10];
		AtCapSorterCycleTime[1];
///////// KONIEC TEST SYMULACJI CZASU CYKLU SORTERA
END_ACTION

ACTION aP09_CapPuttedCheck:
(***********P09_CapPuttedCheck*****************************)
(***********************************************************)
(*******************SPRAWDZANIE NASADEK*********************)
(***********************************************************)	
IF eBeforeScrewers2PackageState[2].bCapPutted THEN
	FOR ic1 := 1 TO 100 DO	
		 IF eBeforeScrewers2PackageState[2].nCardNumber = eRFID[ic1].nCardNumber THEN
			cpc:=ic1;
			
				IF bCapPuttedCheckEnable THEN  
					eRFID[cpc].bFormPresent := TRUE;
					
					eRFID[cpc].bCapOK := eBeforeScrewers2PackageState[2].bCapOK ;
					eRFID[cpc].bCapPutted := eBeforeScrewers2PackageState[2].bCapPutted;
					eRFID[cpc].bCapChecked := eBeforeScrewers2PackageState[2].bCapChecked;	
					IF eBeforeScrewers2PackageState[2].bCapOK THEN						
						eRFID[cpc].bBottlePresent := TRUE;							
					END_IF							
								
					EXIT;	
				ELSE
				eRFID[cpc].bCapOK 		:= eBeforeScrewers2PackageState[2].bCapOK := TRUE;
				eRFID[cpc].bCapChecked	:= eBeforeScrewers2PackageState[2].bCapChecked := TRUE;	
			END_IF
		END_IF	
	END_FOR
END_IF	

IF eBeforeScrewers2PackageState[1].bCapPutted THEN
	FOR ic1 := 1 TO 100 DO
		IF eBeforeScrewers2PackageState[1].nCardNumber = eRFID[ic1].nCardNumber THEN
			cpc:=ic1;
			
				IF bCapPuttedCheckEnable THEN  
				eRFID[cpc].bFormPresent := TRUE;
				
				eRFID[cpc].bCapOK := eBeforeScrewers2PackageState[1].bCapOK ;
				eRFID[cpc].bCapPutted := eBeforeScrewers2PackageState[1].bCapPutted;
				eRFID[cpc].bCapChecked := eBeforeScrewers2PackageState[1].bCapChecked;	
				IF eBeforeScrewers2PackageState[1].bCapOK THEN						
					eRFID[cpc].bBottlePresent := TRUE;							
				END_IF		

		
				EXIT;	
			ELSE
				eRFID[cpc].bCapOK		:= eBeforeScrewers2PackageState[1].bCapOK := TRUE;
				eRFID[cpc].bCapChecked	:= eBeforeScrewers2PackageState[1].bCapChecked := TRUE;	
			END_IF
		END_IF	
	END_FOR
END_IF
(***********************************)
(***********************************)
END_ACTION

ACTION aP10_GripperScrewer:
(***P10_GripperScrewer******)
//Liczenie cykli 
tonAfterScreweEmpty							(IN:=NOT eAfterScrewerPackageState[1].bFormPresent AND NOT eAfterScrewerPackageState[2].bFormPresent,	PT:=T#10MS);


tonCapCorrectCheckAfterScrewerFormSensor.PT	:= T#350MS;
IF bFormTransportersDispencerSlowSpeed THEN
	tonCapCorrectCheckAfterScrewerFormSensor.PT:=T#700MS;
END_IF
(*tonCapCorrectCheckAfterScrewerFormSensor.IN	:= NOT P11_CapCorrectCheck.IbCapCorrectCheckAfterScrewerFormSensor AND 
											NOT P11_CapCorrectCheck.IbCapCorrectCheckFormSensor;//bylo 10 dp było 50 MK dodany czujnik ze sprawdzania nakrętki
tonCapCorrectCheckAfterScrewerFormSensor();		*)
tonCapCorrectCheckAfterScrewerFormSensor	(IN:=	NOT P11_CapCorrectCheck.IbCapCorrectCheckFormSensor, PT:=T#0MS);	//bylo 300						
tofCapCorrectCheckAfterScrewerFormSensor	(IN:=	NOT P11_CapCorrectCheck.IbCapCorrectCheckFormSensor, PT:=T#500MS);							

																				
fbbCapCorrectCheckAfterScrewerFormSensor	(bIN:=
												NOT P11_CapCorrectCheck.IbCapCorrectCheckAfterScrewerFormSensor AND NOT P11_CapCorrectCheck.IbCapCorrectCheckDialAfterScrewerFormSensor
												,tFilterTimeOn:=T#2MS, tFilterTimeOff:=T#0MS, bOUT=> ); //200,0
												
tonThirdFormsSensor							(IN:=P10_GripperScrewer.IbGripperScrewersThirdFormCheckFormSensor, 										PT:=T#20MS);//bylo 100


fbIbGripperScrewersThirdFormCheckFormSensor	(bIN:=
												P10_GripperScrewer.IbGripperScrewersThirdFormCheckFormSensor	AND
												eBeforeScrewersPackageState[1].bFormPresent						AND 
												eBeforeScrewersPackageState[2].bFormPresent						AND 
												eBeforeScrewers2PackageState[1].bFormPresent,
												tFilterTimeOn:=T#35MS(*było250ms*) , tFilterTimeOff:=T#35MS, bOUT=> ); //bylo 20 i przy tym czasie zle filtrowało

fbIbGripperScrewersBeforeThirdFormCheckFormSensor(bIN:=
												P10_GripperScrewer.IbGripperScrewersBeforeThirdFormCheckFormSensor
												,tFilterTimeOn:=T#20MS, tFilterTimeOff:=T#20MS, bOUT=> ); //Czujnik za 3 fo
												
tofFormsDragingPneumaticStationDraged		(IN:=P10_GripperScrewer.fbGripperScrewersDragStation.eRunningState = E_DragStationState.eDraged,	PT:=T#500MS);
tofFormsDragingPneumaticStationDraged.Q;
tofFormsDragingPneumaticStationDraged.PT;
bScrewersReady:=	(NOT bGripperScrewer1Enable OR P10_GripperScrewer.fb2GripperScrewer1.eState = E_Station.eReady AND NOT P10_GripperScrewer.fb2GripperScrewer1.bRun1) AND
					(NOT bGripperScrewer2Enable OR P10_GripperScrewer.fb2GripperScrewer2.eState = E_Station.eReady AND NOT P10_GripperScrewer.fb2GripperScrewer2.bRun1) AND
					(P10_GripperScrewer.fbGripperScrewer1CatchStation.eState=E_Station.eReady AND NOT P10_GripperScrewer.fbGripperScrewer1CatchStation.bCycleDone) AND
					(P10_GripperScrewer.fbGripperScrewer2CatchStation.eState=E_Station.eReady AND NOT P10_GripperScrewer.fbGripperScrewer2CatchStation.bCycleDone)
					AND tonDelayAfterStart.Q;
			
(**** Rozpoczynanie cyklu ***)
//Dojechanie do pełna formatkami przed zakręcarką i ustawienie rejestru, dlatego że zależnie od ilości
//formatek jest różna ilość formatek przed zakręcarkami		
//Kasowanie bitu w PackML Idle	
bDelayAfterStartFullRegister;
IF tonDelayAfterStart.Q AND fb2IbCapPuttedCheckFormSensor.bOUT AND NOT bDelayAfterStartFullRegister THEN
		eBeforeCapControlPackageState[1].bFormPresent	:= TRUE;
		eBeforeScrewers2PackageState[2].bFormPresent	:= TRUE;
		eBeforeScrewers2PackageState[1].bFormPresent	:= TRUE;
		eBeforeScrewersPackageState[2].bFormPresent		:= TRUE;
		eBeforeScrewersPackageState[1].bFormPresent		:= TRUE;
		bDelayAfterStartFullRegister					:= TRUE;
END_IF
			
			
//Przygotowanie do przeciągniecia		
(*IF	bBottleDragingEnable AND 	
								fbIbGripperScrewersThirdFormCheckFormSensor.bOut AND 
								tonDelayAfterStart.Q AND 

								bDelayAfterStartFullRegister AND 
								NOT (P00_PackML.fbPMLAuto.ePMLState = E_PMLState.ePMLState_STOPPING) THEN

	GVL.bBottleDragingStationPrepareRun:=TRUE;
ELSE 
	GVL.bBottleDragingStationPrepareRun:=FALSE;
END_IF*)
(*
IF	bBottleDragingStationEnable AND 	
								NOT fbIbGripperScrewersBeforeThirdFormCheckFormSensor.bOUT AND //Czujnik za 3 formatka (przeciw wypadajacym nakrętkom)	
								fbIbGripperScrewersThirdFormCheckFormSensor.bOut AND 
								tonDelayAfterStart.Q AND 
								bDelayAfterStartFullRegister AND 
								NOT GVL.bBottleDragingStationPrepareRun
THEN
	GVL.bBottleDragingStationPrepareRun:=TRUE;
END_IF*)

	
IF	bBottleDragingStationEnable AND
	//fbIbGripperScrewersThirdFormCheckFormSensor.bOut AND
	P10_GripperScrewer.fbGripperScrewersDragStation.eState = E_Station.eReady AND
	NOT (P00_PackML.fbPMLAuto.ePMLState = E_PMLState.ePMLState_STOPPING) 
THEN
	GVL.bBottleDragingStationPrepareRun						:= TRUE;
END_IF



IF (P00_PackML.fbPMLAuto.ePMLState = E_PMLState.ePMLState_STOPPING) THEN
	GVL.bBottleDragingStationPrepareRun:=FALSE;
END_IF




P11_CapCorrectCheck.IbCapCorrectCheckAfterScrewerFormSensor;

	
CASE iScrewerDragCase OF
	
	0:
		IF GVL.bBottleDragingStationEnable THEN
			iScrewerDragCase				:=	10;
		END_IF
		
	10: //Sprawdzanie czy są formatki przed i spowałniacz gotowy
		IF  (eBeforeScrewersPackageState[1].bFormPresent AND eBeforeScrewersPackageState[2].bFormPresent AND eBeforeScrewers2PackageState[1].bFormPresent) AND
			NOT fbIbGripperScrewersBeforeThirdFormCheckFormSensor.bOUT (*20ms*)
			AND tonThirdFormsSensor.Q (*20ms*)AND (bScrewersReady OR ( NOT bGripperScrewer1Enable AND NOT bGripperScrewer2Enable ))
			AND bDelayAfterStartFullRegister
			AND tonAfterScreweEmpty.Q AND (*rejestry*)
			fbbCapCorrectCheckAfterScrewerFormSensor.bOUT AND // 0ms i 0ms
			NOT (P00_PackML.fbPMLAuto.ePMLState = E_PMLState.ePMLState_STOPPING) AND
			(tonLongDelayFirstDraging.Q OR NOT P11_CapCorrectCheck.IbCapCorrectCheckFormSensor)
			//AND tonCapCorrectCheckAfterScrewerFormSensor.Q (*0ms, bylo 300*) 
			AND (NOT bSingleRealeseIfNoCapFromScrewersDragBlock OR NOT VIS.bSingleRealeseIfNoCapFromScrewers) 
			(*AND bGripperScrewerStoper2ReadyToDrag*)

		THEN 
			VIS.bBottleDragingStationRun	:=	TRUE;
			iScrewerDragCase				:=	20;
		END_IF
		
	20://czy pusto za zakrecarkami 
			iScrewerDragCase:=25;
			
	25: 
		// Reset cyklu jak skonczylo przeciaganie
		IF P10_GripperScrewer.fbGripperScrewersDragStation.bCycleDone THEN
			iScrewerDragCase:=30;
		END_IF
		
		IF NOT VIS.bBottleDragingStationRun THEN
			iScrewerDragCase:=0;
		END_IF
		
	30: // jak skonczylo zakręcanie to wroc do poczatku
//		IF 	(eUnderScrewerPackageState[1].bCapGripperScrewed OR eUnderScrewerPackageState[1].bCapGripperScrewAborted OR NOT eUnderScrewerPackageState[1].bBottlePresent OR NOT eUnderScrewerPackageState[1].bCapOk) AND
//			(eUnderScrewerPackageState[2].bCapGripperScrewed OR eUnderScrewerPackageState[2].bCapGripperScrewAborted OR NOT eUnderScrewerPackageState[2].bBottlePresent OR NOT eUnderScrewerPackageState[2].bCapOk)THEN
			VIS.bBottleDragingStationRun					:=	FALSE;
			GVL.bBottleDragingStationPrepareRun				:=	FALSE;
			iScrewerDragCase								:=	50;
//		END_IF
		
	50:
		IF NOT (P00_PackML.fbPMLAuto.ePMLState = E_PMLState.ePMLState_STOPPING) THEN
			iScrewerDragCase:=0;	
		END_IF
END_CASE

(*nowe*)IF (
(*nowe*)	(eUnderScrewerPackageState[2].bCapGripperScrewed AND NOT eUnderScrewerPackageState[2].bCapGripperScrewAborted) OR
(*nowe*)	NOT eUnderScrewerPackageState[2].bBottlePresent 
(*nowe*)	)
(*nowe*)	AND 
(*nowe*)	iGripperScrewerCase = 5  // Po zakreceniu zapisz czy była butelka zakrecaona czy nie bylo butelki i tylko wtedy wysuwaj szlaban
(*nowe*)THEN
(*nowe*)	bGripperScrewerAcceleratorActuatorTemp := TRUE;
(*nowe*)END_IF
(*nowe*)rtaccelerator 			(CLK:=P10_GripperScrewer.fbGripperScrewersDragStation.eRunningState = E_DragStationState.eEndingOfDrag AND bGripperScrewerAcceleratorActuatorTemp);
tonFormTransporterStop	(IN:=GVL_IO.QbGripperScrewerAcceleratorActuator, PT:=T#150MS);

IF rtaccelerator.q THEN
	GVL_IO.QbGripperScrewerAcceleratorActuator			:=	TRUE;
(*nowe*)	bGripperScrewerAcceleratorActuatorTemp 		:=	FALSE;
ELSIF tonFormTransporterStop.Q THEN
	GVL_IO.QbGripperScrewerAcceleratorActuator	:=	FALSE;
END_IF

//tofScrewerAccelerator	(IN:=(NOT bFormTransportersScrewerStop)
//
//IF P10_GripperScrewer.fbGripperScrewersDragStation.bCycleDone	THEN
//	GVL_IO.QbGripperScrewerAcceleratorActuator:=TRUE;
//END_IF

(************************************)
//zakrecarki
//Deklaracja opóźnienia startu zakręcania
tonStartScrewerDelay();
tonStartScrewerDelay.IN:=	P00_PackML.fbPMLAuto.ePMLState = E_PMLState.ePMLState_EXECUTE AND
							((eUnderScrewerPackageState[1].bFormPresent) AND
							(NOT eUnderScrewerPackageState[1].bCapGripperScrewed AND NOT eUnderScrewerPackageState[1].bCapGripperScrewAborted )) AND
							((eUnderScrewerPackageState[2].bFormPresent) AND 
							(NOT eUnderScrewerPackageState[2].bCapGripperScrewed AND NOT eUnderScrewerPackageState[2].bCapGripperScrewAborted ))
;
tonStartScrewerDelay.PT:=INT_TO_TIME(iGripperScrewerStartDelay + 50);

IF bGripperScrewer1Enable OR bGripperScrewer2Enable THEN
	CASE iGripperScrewerCase OF
		0:
			iGripperScrewerCase	:= 1;
	
		1: //Wykrywanie podjechania nowych wózków i opóźnienie
			IF	tonStartScrewerDelay.Q  THEN	
				iGripperScrewerCase	:= 2;
			END_IF
			
		2:	//Rozpoczecie zakręcania
			IF bGripperScrewer1Enable AND eUnderScrewerPackageState[1].bBottlePresent AND eUnderScrewerPackageState[1].bCapOk  AND eUnderScrewerPackageState[1].nCardNumber > 0 AND 
				(eUnderScrewerPackageState[1].bLidSealed OR NOT bLidFeederEnable) AND
			(eUnderScrewerPackageState[1].bCapSorterPutted AND NOT eUnderScrewerPackageState[1].bCapSorterPuttedAborted OR NOT stCapSorterRead.bEnable)
			 THEN			
				VIS.bGripperScrewer1Run 										:=	NOT bChangeOver;//TRUE;
				bGripperScrewer1Catch											:=	NOT bChangeOver;//TRUE;
			END_IF
				
			IF bGripperScrewer2Enable AND eUnderScrewerPackageState[2].bBottlePresent AND eUnderScrewerPackageState[2].bCapOk  AND eUnderScrewerPackageState[2].nCardNumber > 0 AND
				(eUnderScrewerPackageState[2].bLidSealed OR NOT bLidFeederEnable) AND
			(eUnderScrewerPackageState[2].bCapSorterPutted AND NOT eUnderScrewerPackageState[2].bCapSorterPuttedAborted OR NOT stCapSorterRead.bEnable)
			THEN			
				VIS.bGripperScrewer2Run 										:=	NOT bChangeOver;//TRUE;
				bGripperScrewer2Catch											:=	NOT bChangeOver;//TRUE;
			END_IF
			
			iGripperScrewerCase	:= 3;
			
		3: //Czekanie na koniec zakręcania		
			//Warunek przejścia dalej, albo wykonano zakręcanie albo nie było rozkazu zakręcania (np. brak butelki)
			IF (
				VIS.bGripperScrewer1Run AND (P10_GripperScrewer.fb2GripperScrewer1.bCycleDone1 OR P10_GripperScrewer.fb2GripperScrewer1.bCycleNotDone1)
				OR NOT VIS.bGripperScrewer1Run
				) 
				AND
				(
				VIS.bGripperScrewer2Run AND (P10_GripperScrewer.fb2GripperScrewer2.bCycleDone1 OR P10_GripperScrewer.fb2GripperScrewer2.bCycleNotDone1)
				OR NOT VIS.bGripperScrewer2Run
				)
				THEN
					iGripperScrewerCase	:= 4;
			END_IF
			IF P10_GripperScrewer.fb2GripperScrewer1.eRunningState=E_GripperScrewer.eGoingUp THEN	//Szybsze otwieranie chwytaka
				bGripperScrewer1Catch	:=	FALSE;
			END_IF
			IF P10_GripperScrewer.fb2GripperScrewer2.eRunningState=E_GripperScrewer.eGoingUp THEN	//Szybsze otwieranie chwytaka
				bGripperScrewer2Catch	:=	FALSE;
			END_IF			
		4: //Zapisywanie rejestrów i kasowanie sygnałów

			IF (VIS.bGripperScrewer1Run OR VIS.bGripperScrewer2Run) AND iGripperScrewer1Tool = 0 THEN //tylko dla dwuszczekowej
				VIS.udiGripperScrewerToolCounter := VIS.udiGripperScrewerToolCounter +	1;
			END_IF

			eUnderScrewerPackageState[1].tCapGripperScrewingTime 				:=	P10_GripperScrewer.fb2GripperScrewer1.tCycleTime;
			eUnderScrewerPackageState[2].tCapGripperScrewingTime 				:=	P10_GripperScrewer.fb2GripperScrewer2.tCycleTime;		
			
			IF P10_GripperScrewer.fb2GripperScrewer1.bCycleDone1 THEN
				eUnderScrewerPackageState[1].bCapGripperScrewed 				:=	TRUE;
			ELSIF P10_GripperScrewer.fb2GripperScrewer1.bCycleNotDone1 THEN
				eUnderScrewerPackageState[1].bCapGripperScrewed					:=	FALSE;
				eUnderScrewerPackageState[1].bCapGripperScrewAborted			:=	TRUE;
			ELSIF NOT bGripperScrewer1Enable THEN
				eUnderScrewerPackageState[1].bCapGripperScrewed					:=	TRUE;
			ELSE // Jak wyłączona
				eUnderScrewerPackageState[1].bCapGripperScrewed					:=	TRUE; //dp bylo false
				eUnderScrewerPackageState[1].bCapGripperScrewAborted			:=	TRUE;
			END_IF

			IF P10_GripperScrewer.fb2GripperScrewer2.bCycleDone1 THEN
				eUnderScrewerPackageState[2].bCapGripperScrewed 				:=	TRUE;
			ELSIF P10_GripperScrewer.fb2GripperScrewer2.bCycleNotDone1 THEN
				eUnderScrewerPackageState[2].bCapGripperScrewed					:=	FALSE;
				eUnderScrewerPackageState[2].bCapGripperScrewAborted			:=	TRUE;
			ELSIF NOT bGripperScrewer2Enable THEN
				eUnderScrewerPackageState[2].bCapGripperScrewed					:=	TRUE;
			ELSE // Jak wyłączona
				eUnderScrewerPackageState[2].bCapGripperScrewed					:=	TRUE; //dp bylo false
				eUnderScrewerPackageState[2].bCapGripperScrewAborted			:=	TRUE;
			END_IF
						
			FOR y:=1 TO 100 DO
				IF  eRFID[y].nCardNumber=eUnderScrewerPackageState[1].nCardNumber AND eUnderScrewerPackageState[1].nCardNumber >0 THEN
				 eRFID[y]:=eUnderScrewerPackageState[1];
				 EXIT;
				 END_IF;
			END_FOR
			 
			FOR z:=1 TO 100 DO
				IF  eRFID[z].nCardNumber=eUnderScrewerPackageState[2].nCardNumber AND eUnderScrewerPackageState[2].nCardNumber >0 THEN
					eRFID[z]:=eUnderScrewerPackageState[2];
				 EXIT;
				END_IF;
			END_FOR 
			 	
			 iGripperScrewerCase := 5; 
			 
		5: 
			VIS.bGripperScrewer1Run 											:=	FALSE;	//dp Przeniesione , WAŻNE
			VIS.bGripperScrewer2Run 											:=	FALSE;
			bGripperScrewer1Catch												:=	FALSE;
			bGripperScrewer2Catch												:=	FALSE;

			(***Nie wykonuj dalej ruchu gdy wcisnięty stop lub błąd***)
			IF NOT (P00_PackML.fbPMLAuto.ePMLState = E_PMLState.ePMLState_STOPPING) THEN
				iGripperScrewerCase := 0;
			END_IF
			
	END_CASE
ELSE
	eUnderScrewerPackageState[1].bCapGripperScrewed 				:=	TRUE;
	eUnderScrewerPackageState[2].bCapGripperScrewed 				:=	TRUE;	
	
	FOR y:=1 TO 100 DO
		IF  eRFID[y].nCardNumber=eUnderScrewerPackageState[1].nCardNumber AND eUnderScrewerPackageState[1].nCardNumber >0 THEN
			 eRFID[y]:=eUnderScrewerPackageState[1];
		EXIT;
		END_IF;
	 END_FOR
			 
	FOR z:=1 TO 100 DO
		IF  eRFID[z].nCardNumber=eUnderScrewerPackageState[2].nCardNumber AND eUnderScrewerPackageState[2].nCardNumber >0 THEN
			eRFID[z]:=eUnderScrewerPackageState[2];
		EXIT;
		END_IF;
	END_FOR 
			 
END_IF
END_ACTION

ACTION aP10_GripperScrewerGate:
fbGripperScrewerStoperSensorDelay.bIN := P10_GripperScrewer.fbGripperScrewersDragStation.eRunningState = E_DragStationState.eDraging 
						   AND ((P00_PackML.fbPMLAuto.ePMLState = E_PMLState.ePMLState_STOPPING) OR  (P00_PackML.fbPMLAuto.ePMLState = E_PMLState.ePMLState_EXECUTE));

fbGripperScrewerStoperSensorDelay(tFilterTimeOn:=T#120MS, tFilterTimeOff:=T#20MS);

				   
lrGripperScrewerStoperPosition :=	(188.25 * EXPT(lrBottleDragingStationVelocity,-0.404));


tofQbGripperScrewerStoperActuator	(IN:=fbGripperScrewerStoperSensorDelay.bOUT   AND
									P10_GripperScrewer.fbGripperScrewersDragStation.lrActualDragPosition > (lrGripperScrewerStoperPosition+10) AND 
									P10_GripperScrewer.fbGripperScrewersDragStation.lrActualDragPosition < 100, PT:=T#500MS);
										
QbGripperScrewerStoperActuator		:= tofQbGripperScrewerStoperActuator.Q ;


//Dodatkowy stoper i szlaban

//Wysuniecie Stoper2
rtQbGripperScrewerStoperActuator			(CLK:= P10_GripperScrewer.fbGripperScrewersDragStation.eRunningState  = E_DragStationState.eEndingOfDragDone , Q=>);
IF  rtQbGripperScrewerStoperActuator.Q THEN
	QbGripperScrewerStoper2Actuator				:= TRUE;
END_IF

//Wysuniecie szlaban
fbQbGripperScrewerGateBeforeActuator		(bIN:=		//MAIN.IbCapSorterAfterFormSensor3 AND
													(*NOT*) P09_CapPuttedCheck.IbCapPuttedCheckFormSensor AND
													NOT P10_GripperScrewer.IbGripperScrewersbeforeThirdFormCheckFormSensor AND
														(*P10_GripperScrewer.IbGripperScrewersSixthFormCheckFormSensor AND*)												
														P10_GripperScrewer.IbGripperScrewersThirdFormCheckFormSensor 
													
											,tFilterTimeOn:=T#500MS, tFilterTimeOff:=T#500MS);
rtfbQbGripperScrewerGateBeforeActuator 		(CLK:= fbQbGripperScrewerGateBeforeActuator.bOUT,	Q=>);
QbGripperScrewerGateBeforeActuator 			S= rtfbQbGripperScrewerGateBeforeActuator.Q;
//Schowanie Stoper2
tonQbGripperScrewerGateBeforeActuator		(IN:= QbGripperScrewerGateBeforeActuator,PT:=T#5MS);
IF tonQbGripperScrewerGateBeforeActuator.Q THEN 
	QbGripperScrewerStoper2Actuator				:= FALSE;
END_IF

//Ready do przeciągania
IF tonQbGripperScrewerGateBeforeActuator.Q THEN 
	bGripperScrewerStoper2ReadyToDrag			:= TRUE;
END_IF

// Koniec przeciągania
IF P10_GripperScrewer.fbGripperScrewersDragStation.eRunningState = E_DragStationState.eEndingOfDrag THEN
	bGripperScrewerStoper2ReadyToDrag := FALSE;
	//Schowanie szlaban
	QbGripperScrewerGateBeforeActuator:= FALSE;
END_IF


//Koniec Dodatkowy stoper i szlaban
END_ACTION

ACTION aP11_CapCorrectCheck:
(***********P11_CapCorrectCheckCamera*****************************)
(*****************************************************************)

eUnderCorrectCapPackageState[1].bCapCorrectCheckCameraOK;		
eUnderCorrectCapPackageState[1].bCapCorrectCheckCameraChecked;


(*********************P11_CapCorrectCheck*******************)
(***********************************************************)
(*******************SPRAWDZANIE ZAKRECANIA******************)
(***********************************************************)	
tofIbCapCorrectCheckFormSensor(IN:=P11_CapCorrectCheck.IbCapCorrectCheckFormSensor,PT:=T#0MS);
rttofIbCapCorrectCheckFormSensor(CLK:=tofIbCapCorrectCheckFormSensor.Q, Q=>);
//IF P11_CapCorrectCheck.IbCapCorrectCheckFormSensor THEN 
IF tofIbCapCorrectCheckFormSensor.Q THEN 
	IF rttofIbCapCorrectCheckFormSensor.Q THEN // do usun
		eUnderCorrectCapPackageState[1].bBottlePresent						:=	FALSE;
	END_IF
	IF 	P11_CapCorrectCheck.IbCapCorrectCheckBottleSensor	THEN 						// Dodatkowe sprawdzanie butelki
		eUnderCorrectCapPackageState[1].bBottlePresent						:=	TRUE;	
		bCapCorrectCheckBottleSensorLast									:=	TRUE;
	END_IF				
	(*Kasowanie butelki*)
	//IF eUnderCorrectCapPackageState[1].bBottlePresent AND NOT P11_CapCorrectCheck.IbCapCorrectCheckFormSensor AND NOT bCapCorrectCheckBottleSensorLast THEN
	//	eUnderCorrectCapPackageState[1].bBottlePresent						:=	FALSE;
	//	iCapCorrectCheckBottleSensorLast	:=	iCapCorrectCheckBottleSensorLast +1;
	//END_IF
	(*Koniec Kasowanie butelki*)

	IF P11_CapCorrectCheck.eCapCorrectCheckRunningState = E_CheckerState.eCapOK THEN	// Jeżeli czujnik wykrył nasadki			
		eUnderCorrectCapPackageState[1].bCapCorrectCapOn					:=	TRUE;
		eUnderCorrectCapPackageState[1].bCapCorrectNOK						:=	FALSE;
		eUnderCorrectCapPackageState[1].bBottlePresent						:=	TRUE;								
	END_IF
	IF P11_CapCorrectCheck.eCapCorrectCheckRunningState = E_CheckerState.eCapNOK THEN	// Jeżeli czujnik wykrył zle zakręcenie				
		eUnderCorrectCapPackageState[1].bCapCorrectNOK						:=	TRUE;
		eUnderCorrectCapPackageState[1].bCapCorrectCapOn					:=	TRUE;
		eUnderCorrectCapPackageState[1].bBottlePresent						:=	TRUE;
	END_IF
	IF NOT bCapCorrectCheckEnable THEN
		eUnderCorrectCapPackageState[1].bCapCorrectCapOn					:=	TRUE;
		eUnderCorrectCapPackageState[1].bCapCorrectNOK						:=	FALSE;	
	END_IF	
	
	eUnderCorrectCapPackageState[1].bCapCorrectChecked						:=	TRUE; 	// Ustawienie że było sprawdzanie

	IF NOT bCapCorrectCheckCameraEnable THEN											// Wylaczony czujnik wizyjny
		IF eUnderCorrectCapPackageState[1].bBottlePresent	THEN	
			eUnderCorrectCapPackageState[1].bCapCorrectCheckCameraOK		:=	TRUE;
			eUnderCorrectCapPackageState[1].bCapCorrectCheckCameraChecked	:=	FALSE;
		END_IF
	END_IF
												
	FOR cch := 1 TO 100 DO															//Przeszukiwanie tablicy RFID
		 IF eUnderCorrectCapPackageState[1].nCardNumber = eRFID[cch].nCardNumber AND eUnderCorrectCapPackageState[1].nCardNumber > 0 THEN	//Jeżeli znaleziono w tablicy takie RFID jak w rejestrze(które zostało przypisane przed zakręcarkami)
			nccc:=cch; eRFID[nccc].bCapCorrectCapOn; eRFID[nccc].bCapCorrectNOK; eRFID[nccc].bCapCorrectChecked; 
			
			nUnderCorrectCapPackageStateLastnCardNumber						:=	eRFID[cch].nCardNumber;	                                              					
			eRFID[cch].bCapCorrectCapOn										:=	eUnderCorrectCapPackageState[1].bCapCorrectCapOn;	
			eRFID[cch].bCapCorrectNOK										:=	eUnderCorrectCapPackageState[1].bCapCorrectNOK	;
			IF 	eUnderCorrectCapPackageState[1].bBottlePresent THEN
				eRFID[cch].bBottlePresent									:=	TRUE;
			//ELSE								(*Kasowanie butelki*) //nie sprawdza sie
			//	eRFID[cch].bBottlePresent									:=	FALSE; //dp do testów
			END_IF										
		
			
			eRFID[cch].bCapCorrectChecked									:=	eUnderCorrectCapPackageState[1].bCapCorrectChecked;						
			eRFID[cch].bCapCorrectCheckCameraOK								:=	eUnderCorrectCapPackageState[1].bCapCorrectCheckCameraOK;
			eRFID[cch].bCapCorrectCheckCameraChecked						:=	eUnderCorrectCapPackageState[1].bCapCorrectCheckCameraChecked;
			(*Spowalnianie transportera*)
			IF (eRFID[cch].bBottlePresent AND NOT eRFID[cch].bCapOK AND NOT bROPPFeederEnable) OR
 				(eRFID[cch].bBottlePresent AND NOT eRFID[cch].bROPPCappingOK AND  bROPPFeederEnable) 
				THEN
				ulFormTransportersScrewerSlowNumber							:=	eRFID[cch].nCardNumber;
				bFormTransportersDispencerSlowSpeedPulse					:=	TRUE;
				bFormTransportersDispencerResetSpeed						:=	FALSE;
				iFormTransportersScrewerResetSpeedPulse						:=	iFormTransportersScrewerResetSpeedPulse	+	1;
			END_IF
			EXIT;
		END_IF
	END_FOR		
ELSE
	bCapCorrectCheckBottleSensorLast										:=	FALSE;
END_IF


rtP11_CapCorrectCheckfbCapCorrectCheckCamerabCycleDone	(CLK:=P11_CapCorrectCheck.eCapCorrectCheckCameraRunningState = E_CheckerState.eLidOK OR P11_CapCorrectCheck.eCapCorrectCheckCameraRunningState =  E_CheckerState.eLidNOK,	Q=>);
IF rtP11_CapCorrectCheckfbCapCorrectCheckCamerabCycleDone.Q AND bCapCorrectCheckCameraEnable THEN
	
	nUnderCorrectCapPackageStateLastnCardNumber;
	FOR cchc := 1 TO 100 DO	

		 IF eRFID[cchc].nCardNumber = nUnderCorrectCapPackageStateLastnCardNumber THEN	

			IF P11_CapCorrectCheck.eCapCorrectCheckCameraRunningState = E_CheckerState.eLidOK THEN // Jeżeli kamera wykryła dobre ustawienie butelki			
				eRFID[cchc].bCapCorrectCheckCameraOK		:=	TRUE;
				eRFID[cchc].bCapCorrectCheckCameraChecked	:=	FALSE;
				nCapCorrectCheckCameraOK	:=	nCapCorrectCheckCameraOK	+	1;			
			END_IF
			
			IF P11_CapCorrectCheck.eCapCorrectCheckCameraRunningState =  E_CheckerState.eLidNOK THEN // Jeżeli kamera wykryła zle ustawienie butelki				
				eRFID[cchc].bCapCorrectCheckCameraOK		:=	FALSE;
				eRFID[cchc].bCapCorrectCheckCameraChecked	:=	TRUE;
				nCapCorrectCheckCameraNOK	:=	nCapCorrectCheckCameraNOK	+	1;
				
				IF NOT P11_CapCorrectCheck.IbCapCorrectCheckCameraLogic1CapPresent THEN
					eRFID[cchc].bCapCorrectCapOn	:=	FALSE;
				END_IF
				
			END_IF
			
		END_IF
	END_FOR
	
END_IF

(***********************************************************)
(***********************************************************)
END_ACTION

ACTION aP13_BottleTransfer:
(*
Nazwa:			aP13_BottleTransfer
Opis:			Przenoszenie opakowań na etykiaciarke i wagę
Wersja:			v0.12
Data:			2025-08-19
Autor:			DJ,DP,MP
Urzadzenia:		
Konfiguracja:	
Info:
- [20250819] [DP] - Przeniesione liczniki
- [20240925] [DP] - Rotate i KTP
*)



(*******************TRANSFER BUTELEK**********************)
(*********************************************************)

//Opoźnienie odczytania
tonReadedCardFirstDelayBottleTransfer			(IN:=eRobotPackageState[1].nCardNumber >0 AND eRobotPackageState[1].bFormPresent AND P13_BottleTransfer.IbFirstFormCheckFormSensor,PT:=T#100MS);//Bylo dp1 50 Tutaj musi być jakieś opóźnienie bo zdarza się
tonReadedCardSecondDelayBottleTransfer			(IN:=eRobotPackageState[2].nCardNumber >0 AND eRobotPackageState[2].bFormPresent AND P13_BottleTransfer.IbSecondFormCheckFormSensor,PT:=T#100MS);//Bylo dp1 50 Tutaj musi być jakieś opóźnienie bo zdarza się
tonNotReadedCardFirstDelayBottleTransfer		(IN:=eRobotPackageState[1].nCardNumber =0 AND eRobotPackageState[1].bFormPresent AND P13_BottleTransfer.IbFirstFormCheckFormSensor,PT:=T#3S);//Tutaj musi być jakieś opóźnienie bo zdarza się
tonNotReadedCardSecondDelayBottleTransfer		(IN:=eRobotPackageState[2].nCardNumber =0 AND eRobotPackageState[2].bFormPresent AND P13_BottleTransfer.IbSecondFormCheckFormSensor,PT:=T#3S);//Tutaj musi być jakieś opóźnienie bo zdarza się
fbIbBottleTransferFormAfterSensor				(bIN:=P13_BottleTransfer.IbBottleTransferFormAfterSensor AND P13_BottleTransfer.IbBottleTransferFormAfterSensor2,	tFilterTimeOn:=T#30MS,	tFilterTimeOff:=T#500MS); //bylo na on 500

(*Przejazd przez wagę co którąś butelkę*)
(*IF iBottleTransferWeightInterval < 5 THEN
	iBottleTransferWeightInterval := 100;
END_IF*)
IF NOT bBottleTransferWeightEnable THEN
	udiBottleTransferWeightIntervalCount := 0;
END_IF
//Pierwsze przepisanie
IF bBottleTransferWeightEnable AND udiBottleTransferWeightIntervalCount = 0 THEN
	udiBottleTransferWeightIntervalCount := VIS.udiCounterGlobal;
END_IF
// Wystawienie sygnału do połóżenia na wagę
IF bBottleTransferWeightEnable AND NOT bBottleTransferDoWeight AND iBottleTransferCase = 0 AND (VIS.udiCounterGlobal >= (udiBottleTransferWeightIntervalCount + INT_TO_UDINT(iBottleTransferWeightInterval)) OR VIS.bBottleTransferForceWeight) THEN
	bBottleTransferDoWeight := TRUE;
END_IF
	
(*Dodane do testów czy problem z RFID czy przesuwaniem rejestru*)
rttonNotReadedCardFirstDelayBottleTransfer(CLK:=tonNotReadedCardFirstDelayBottleTransfer.Q);
rttonNotReadedCardSecondDelayBottleTransfer(CLK:=tonNotReadedCardSecondDelayBottleTransfer.Q);
	
IF rttonNotReadedCardFirstDelayBottleTransfer.Q THEN
	iCounterRepairNotReadedFirst:= iCounterRepairNotReadedFirst+1;
END_IF

	
IF rttonNotReadedCardSecondDelayBottleTransfer.Q THEN
	iCounterRepairNotReadedSecond:= iCounterRepairNotReadedSecond+1;
END_IF
(*Dodane do testów czy problem z RFID czy przesuwaniem rejestru*)

tonCycleLabelMachineFullSensor					(IN:=(NOT P16_LabelMachine.IbLabelMachineFullSensor) (*AND (P16_LabelMachine.IbLabelMachineWorking OR NOT bLabelMachineEnable)*),PT:=T#10MS);//bylo 200


tonCycleBadBottleConveyorFullSensor				(IN:=P14_BadBottleConyevor.IbBadBottleConveyorFullSensor ,PT:=T#1S);//bylo 200
tonCycleBadBottleConveyorFullSensor2			(IN:=P14_BadBottleConyevor.IbBadBottleConveyorFullSensor ,PT:=T#5S);//bylo 200

// Czekaj aż dojedzenie druga formatka
tonWaitUntilSecondFormPresent(IN:= 		P13_BottleTransfer.IbSecondFormCheckFormSensor  AND P01_Gates.QbBottleTransferGate1Actuator AND
										tonDelayAfterStart.Q AND
										eRobotPackageState[1].bFormPresent 
									AND eRobotPackageState[2].bFormPresent AND
									NOT eRobotPackageState[2].bBottleTransferedToExit AND NOT eRobotPackageState[2].bBottleTransferedToLabeler AND
									NOT eRobotPackageState[1].bBottleTransferedToExit AND NOT eRobotPackageState[1].bBottleTransferedToLabeler 
									, PT:=T#300MS); //bylo 400 600ms
									
(*Spowalnianie transportera*)									
IF bFormTransportersDispencerSlowSpeed THEN
	tonWaitUntilSecondFormPresent(IN:=P13_BottleTransfer.IbSecondFormCheckFormSensor AND P01_Gates.QbBottleTransferGate1Actuator AND
									 		tonDelayAfterStart.Q AND
											eRobotPackageState[1].bFormPresent 
										AND eRobotPackageState[2].bFormPresent AND
										NOT eRobotPackageState[2].bBottleTransferedToExit AND NOT eRobotPackageState[2].bBottleTransferedToLabeler AND
										NOT eRobotPackageState[1].bBottleTransferedToExit AND NOT eRobotPackageState[1].bBottleTransferedToLabeler 
										, PT:=T#700MS);	//bylo 1000
END_IF
						
			
tonWaitUntilSecondFormPresent.Q;

nVarModuloSimulation:= MAIN.iCountSimulation MOD 25;

(*Wlaczenie tylko inkjetowanie, traktowanie wszystkich formatek jako z butelkami i dobre*)
IF VIS.bBottleTransferAllFormsToLabeler  THEN
	eRobotPackageState[1].bBottlePresent		:= 	TRUE;
	eRobotPackageState[1].bDosed				:= 	TRUE;	
	eRobotPackageState[1].bWeightOK 			:= 	TRUE;
    eRobotPackageState[1].bCapOK 				:= 	TRUE;
	eRobotPackageState[1].bCapGripperScrewed 	:=	TRUE;
	eRobotPackageState[1].bCapCorrectCapOn		:=	TRUE;
	eRobotPackageState[2].bBottlePresent		:= 	TRUE;
	eRobotPackageState[2].bDosed				:= 	TRUE;	
	eRobotPackageState[2].bWeightOK 			:= 	TRUE;
    eRobotPackageState[2].bCapOK 				:= 	TRUE;
	eRobotPackageState[2].bCapGripperScrewed 	:=	TRUE;
	eRobotPackageState[2].bCapCorrectCapOn		:=	TRUE;
END_IF

IF NOT bCapCorrectCheckEnable THEN 
	eRobotPackageState[2].bCapCorrectCapOn		:=	TRUE;
	eRobotPackageState[1].bCapCorrectCapOn		:=	TRUE;
END_IF

IF NOT bCapCorrectCheckCameraEnable THEN 
	eRobotPackageState[2].bCapCorrectCheckCameraOK	:=	TRUE;
	eRobotPackageState[1].bCapCorrectCheckCameraOK	:=	TRUE;
END_IF
	
(*Przenoszenie wszystkich do wyyjscia, bez robota*)
IF VIS.bBottleTransferAllFormsToExit THEN
	eRobotPackageState[1].bBottlePresent		:= 	TRUE;
	eRobotPackageState[2].bBottlePresent		:= 	TRUE;
END_IF

IF tonReadedCardFirstDelayBottleTransfer.Q THEN
	bRobotCycleRFIDReadedOne					:=	TRUE; //Zapisanie że przeczytało RFID
ELSE
	bRobotCycleRFIDReadedOne					:=	FALSE; //Zapisanie że nieprzeczytało RFID
END_IF;

IF tonReadedCardSecondDelayBottleTransfer.Q THEN
	bRobotCycleRFIDReadedTwo					:=	TRUE; //Zapisanie że przeczytało RFID
ELSE
	bRobotCycleRFIDReadedTwo					:=	FALSE; //Zapisanie że nieprzeczytało RFID
END_IF;	

//ładowanie ilości formatek do wyjazdu
//w1
//ctdCounterFormOnRobot				(CD:=MAIN.ftfbIbFirstFormCheckFormSensor.Q,  PV:=INT_TO_WORD(nCounterFormsToLoad),Q=>,CV=>); //zb opad
//w2
//IF MAIN.ftfbIbFirstFormCheckFormSensor.Q THEN
IF MAIN.ftfbIbFirstFormCheckFormSensor.Q THEN	
	nCounterFormsToLoad;
	nCounterForms	:=	nCounterForms	+	1;
END_IF

//Sprawdzanie czy wszystko ok na pierwszym rejestrze robota
(*bRobotPackageState1OK :=
						(
							(
							eRobotPackageState[1].bBottlePresent 
								(*AND eRobotPackageState[1].bDosed*) AND eRobotPackageState[1].bWeightOK AND eRobotPackageState[1].bCapOK AND eRobotPackageState[1].bCapCorrectCapOn 
                        		AND NOT eRobotPackageState[1].bCapCorrectNOK AND (eRobotPackageState[1].bCapGripperScrewed AND NOT eRobotPackageState[1].bCapGripperScrewAborted)
							) OR 
							(VIS.bBottleTransferAllFormsToLabeler AND NOT (VIS.bSimulation AND  nVarModuloSimulation=0 ))
						) AND NOT VIS.bBottleTransferAllFormsToExit AND bRobotCycleRFIDReadedOne;			
						
//Sprawdzanie czy coś jest źle  na pierwszym rejestrze robota		
bRobotPackageState1NOK := ((
							(	
								(
									eRobotPackageState[1].bBottlePresent AND
									( 
										(*NOT eRobotPackageState[1].bDosed OR*) NOT eRobotPackageState[1].bWeightOK OR NOT eRobotPackageState[1].bCapOK OR NOT eRobotPackageState[1].bCapCorrectCapOn OR eRobotPackageState[1].bCapCorrectNOK OR 
						 			  	NOT eRobotPackageState[1].bCapGripperScrewed OR eRobotPackageState[1].bCapGripperScrewAborted
									)
								) 
								OR	VIS.bBottleTransferAllFormsToExit
							) AND NOT VIS.bBottleTransferAllFormsToLabeler
						) (**)OR tonNotReadedCardFirstDelayBottleTransfer.Q(**)) OR (VIS.bSimulation AND  nVarModuloSimulation=0 ); //przeniesiony NOTreaded do Empty
						
					


bRobotPackageState1Empty	:= (NOT eRobotPackageState[1].bBottlePresent AND bRobotCycleRFIDReadedOne) (*OR tonNotReadedCardFirstDelayBottleTransfer.Q*);*)
bRobotPackageState1OK :=
						(
							(
							eRobotPackageState[1].bBottlePresent 
							AND ((eRobotPackageState[1].bROPPPutted AND eRobotPackageState[1].bROPPCapped AND eRobotPackageState[1].bROPPCappingOK) OR NOT bROPPCappingEnable)
								(**)AND eRobotPackageState[1].bDosed(**) AND eRobotPackageState[1].bWeightOK AND eRobotPackageState[1].bCapOK AND eRobotPackageState[1].bCapCorrectCapOn AND 
                        		NOT eRobotPackageState[1].bCapCorrectNOK AND (eRobotPackageState[1].bCapGripperScrewed AND NOT eRobotPackageState[1].bCapGripperScrewAborted)
							) OR 
							(VIS.bBottleTransferAllFormsToLabeler AND NOT (VIS.bSimulation AND  nVarModuloSimulation=0 ))
						) AND NOT VIS.bBottleTransferAllFormsToExit AND bRobotCycleRFIDReadedOne;			
						
//Sprawdzanie czy coś jest źle  na pierwszym rejestrze robota		
bRobotPackageState1NOK := ((
							(									
								eRobotPackageState[1].bBottlePresent AND NOT bRobotPackageState1OK
								OR	VIS.bBottleTransferAllFormsToExit
							) AND NOT VIS.bBottleTransferAllFormsToLabeler
						) OR tonNotReadedCardFirstDelayBottleTransfer.Q) OR (VIS.bSimulation AND  nVarModuloSimulation=0 ); 
									


bRobotPackageState1Empty	:= (NOT eRobotPackageState[1].bBottlePresent AND bRobotCycleRFIDReadedOne) (*OR tonNotReadedCardFirstDelayBottleTransfer.Q*);
bRobotPackageState2OK := 
						(
							(
							eRobotPackageState[2].bBottlePresent 
							AND ((eRobotPackageState[2].bROPPPutted AND eRobotPackageState[2].bROPPCapped AND eRobotPackageState[2].bROPPCappingOK) OR NOT bROPPCappingEnable)
							(**)AND eRobotPackageState[2].bDosed(**) AND eRobotPackageState[2].bWeightOK AND eRobotPackageState[2].bCapOK AND eRobotPackageState[2].bCapCorrectCapOn AND 
					    	 NOT eRobotPackageState[2].bCapCorrectNOK AND (eRobotPackageState[2].bCapGripperScrewed	AND NOT eRobotPackageState[2].bCapGripperScrewAborted)
						) OR 
        				 VIS.bBottleTransferAllFormsToLabeler
						) AND NOT VIS.bBottleTransferAllFormsToExit AND bRobotCycleRFIDReadedTwo ;
						 
						 
//Sprawdzanie czy coś jest źle  na drugim rejestrze robota			
bRobotPackageState2NOK := 
						(
							 (
									eRobotPackageState[2].bBottlePresent AND NOT bRobotPackageState2OK 
									 OR	 VIS.bBottleTransferAllFormsToExit
							) AND NOT VIS.bBottleTransferAllFormsToLabeler
						) OR tonNotReadedCardSecondDelayBottleTransfer.Q;

bRobotPackageState2Empty	:= (NOT eRobotPackageState[2].bBottlePresent AND bRobotCycleRFIDReadedTwo) (*OR tonNotReadedCardSecondDelayBottleTransfer.Q*);	
//Sprawdzanie czy wszystko ok na drugim rejestrze robota
(*bRobotPackageState2OK := ((eRobotPackageState[2].bBottlePresent (*AND eRobotPackageState[1].bDosed*) AND eRobotPackageState[2].bWeightOK AND eRobotPackageState[2].bCapOK AND eRobotPackageState[2].bCapCorrectCapOn AND 
					     NOT eRobotPackageState[2].bCapCorrectNOK AND (eRobotPackageState[2].bCapGripperScrewed	AND NOT eRobotPackageState[2].bCapGripperScrewAborted)) OR 
        				 VIS.bBottleTransferAllFormsToLabeler) AND NOT VIS.bBottleTransferAllFormsToExit AND bRobotCycleRFIDReadedTwo ;
						 
						 
//Sprawdzanie czy coś jest źle  na drugim rejestrze robota			
bRobotPackageState2NOK := (((eRobotPackageState[2].bBottlePresent AND ((*NOT eRobotPackageState[1].bDosed OR*) NOT eRobotPackageState[2].bWeightOK OR NOT eRobotPackageState[2].bCapOK OR NOT eRobotPackageState[2].bCapCorrectCapOn 
						  OR eRobotPackageState[2].bCapCorrectNOK OR NOT eRobotPackageState[2].bCapGripperScrewed OR eRobotPackageState[2].bCapGripperScrewAborted)) OR	
						  VIS.bBottleTransferAllFormsToExit) AND NOT VIS.bBottleTransferAllFormsToLabeler) (**)OR tonNotReadedCardSecondDelayBottleTransfer.Q(**);

bRobotPackageState2Empty	:= (NOT eRobotPackageState[2].bBottlePresent AND bRobotCycleRFIDReadedTwo) (*OR tonNotReadedCardSecondDelayBottleTransfer.Q*);						  
*)
					  

////////////////////////////////////////////////////////////////////////	
// dodane 06.08 Damian na testy zliczania błędnie odrzucony					  

// jedna butelka była zła
rtbRobotPackageState1NOK(CLK:=bRobotPackageState1NOK);					
						
IF rtbRobotPackageState1NOK.Q THEN
	ibRobotPackageState1NOK:=ibRobotPackageState1NOK+1;
END_IF
	
// dwie butelki były złe
rtbRobotPackageState2NOK(CLK:=bRobotPackageState2NOK AND bRobotPackageState1NOK);					
						
IF rtbRobotPackageState2NOK.Q THEN
	ibRobotPackageState2NOK:=ibRobotPackageState2NOK+1;
END_IF


///////////////////////////////////////////////////////
// sprawdzanie czy butelka do obrocenia
bRobotPackageState1Rotate	:= ((eRobotPackageState[1].bBottlePresent AND NOT eRobotPackageState[1].bCapCorrectCheckCameraOK AND eRobotPackageState[1].bCapCorrectCheckCameraChecked))
                         	AND bRobotPackageState1OK AND bCapCorrectCheckCameraEnable;
bRobotPackageState2Rotate	:= ((eRobotPackageState[2].bBottlePresent AND NOT eRobotPackageState[2].bCapCorrectCheckCameraOK AND eRobotPackageState[2].bCapCorrectCheckCameraChecked))
                         	AND bRobotPackageState2OK AND bCapCorrectCheckCameraEnable;

///////////////////////////////////////////////////////

CASE iBottleTransferCase OF
	
	0: //KASOWANIE WSZYSTKICH ROZKAZÓW
		bRobotStationDone						:=	FALSE;
		VIS.bBottleTransferRun 					:=	FALSE;
		VIS.bGateRobotEntranceRun 				:=	FALSE;
		bRobotGateStayOpen						:= 	FALSE;
		iRobotPickCase							:=	0; 
		iBottleTransferCase 					:=	1; 
		
	1: // CZEKANIE NA FORMATKE I WYKONANIE RUCHU ROBOTA JAK SIĘ POJAWI

					CASE iRobotPickCase OF 
						
						0:	
								//Jak robot włączony to idz do sprawdzania formatek
								IF P13_BottleTransfer.fbBottleTransfer.eState = E_Station.eReady AND NOT bChangeOver THEN	
									iRobotPickCase					:=10;
								END_IF
								
								//Jak robot wyłączony to do wyjazdu i otwarcia szlabanu
								IF P13_BottleTransfer.fbBottleTransfer.eState = E_Station.eDisabled OR bChangeOver THEN	
									iRobotPickCase					:=220;
								END_IF
								
						10:		
								//Są dwie formatk
								IF tonWaitUntilSecondFormPresent.Q AND (NOT (P00_PackML.fbPMLAuto.ePMLState = E_PMLState.ePMLState_STOPPING) OR P11_CapCorrectCheck.IbCapCorrectCheckAfterScrewerFormSensor) THEN									
									iRobotPickCase				:= 20;
									(***Zapisywanie który numer formatki w tablicy RFID trzeba wyczyścić***)
									bRFIDClearAfterRobot			:=		TRUE;
									(***Koniec Zapisywanie który numer formatki w tablicy RFID trzeba wyczyścić***)				
								END_IF	
								
						20:
								// 2 Formatki OK [OK]
								IF	bRobotPackageState1OK AND bRobotPackageState2OK AND 
									(
									(bRobotPackageState1Rotate AND bRobotPackageState2Rotate) OR 
									(NOT bRobotPackageState1Rotate AND NOT bRobotPackageState2Rotate) 
									) AND  
									NOT bBottleTransferDoWeight THEN 
									
									nCounterCase7						:= nCounterCase7 + 1;
									iRobotPickCase						:= 200;

								// 2 Formatka NOK [OK]
								ELSIF bRobotPackageState1NOK AND bRobotPackageState2NOK THEN 
									bBadBottleConveyorStartTriggerDelay	:= TRUE;
									//bAddBadPackageReason				:= TRUE;
									nCounterCase8						:= nCounterCase8 + 1;
									iRobotPickCase						:= 210;															
										
								//Odczytalo formatki ale pierwsza zła, a druga dobra [OK]
								ELSIF bRobotPackageState1NOK AND bRobotPackageState2OK THEN 
									bBadBottleConveyorStartTriggerDelay	:= TRUE;
									nCounterCase9						:= nCounterCase9 + 1;
									iRobotPickCase						:= 110;	
								//Odczytalo formatki ale druga zła a pierwsza dobra [OK]
								ELSIF (bRobotPackageState1OK OR (bBottleTransferDoWeight AND bRobotPackageState1OK)) AND (bRobotPackageState2NOK OR bBottleTransferDoWeight OR bCapCorrectCheckCameraEnable) THEN 
									
									nCounterCase10						:= nCounterCase10+1;
									iRobotPickCase						:= 100;									

								//Odczytalo formatki ale nie ma 2 butelek [OK]
								ELSIF bRobotPackageState1Empty AND bRobotPackageState2Empty THEN 
									
									nCounterCase11						:= nCounterCase11 + 1;
									iRobotPickCase						:= 220;							
								
								// Odczytalo obydwie ale w drugiej nie ma butelki [OK]
								ELSIF (bRobotPackageState1OK OR (bBottleTransferDoWeight AND bRobotPackageState1OK)) AND bRobotPackageState2Empty THEN 
									
									nCounterCase12						:= nCounterCase12+1;
									iRobotPickCase						:= 100;

								//Odczytalo obydwie ale pierwsza nie ma butelki	[OK]	
								ELSIF bRobotPackageState1Empty AND bRobotPackageState2OK THEN 
									
									nCounterCase13						:= nCounterCase13 + 1;
									iRobotPickCase						:= 120; 
									
								//Pierwsza formatka NOK, 2 formatka EMPTY		
							   ELSIF bRobotPackageState1NOK AND bRobotPackageState2Empty THEN
									bBadBottleConveyorStartTriggerDelay :=TRUE;
									//bAddBadPackageReason				:=	TRUE;
									nCounterCase14						:= nCounterCase14+1;
									iRobotPickCase						:= 110;	
									
								ELSIF bRobotPackageState1Empty AND bRobotPackageState2NOK THEN
									
									nCounterCase15						:= nCounterCase15+1;
									iRobotPickCase						:= 120;
									
								END_IF			
				
							100: //Pobranie i odłozenie jednej butelki na dobre	
									nCheckCountR1:=nCheckCountR1+1;
									VIS.nBottleTransferPickOption			:=	1; // 1 butelka
									VIS.nBottleTransferPlaceOption			:=	1; //Dobre butelki 
									IF bBottleTransferDoWeight AND NOT bRobotPackageState1Rotate THEN
										VIS.nBottleTransferPlaceOption		:=	3; // Przenoszenie na wagę																																						
									END_IF
										
									IF 	bRobotPackageState1Rotate  THEN 	(* OBRÓT CHWYTAKA *)
										VIS.nBottleTransferPlaceOption		:=	4; 
									END_IF	
																										
									IF tonCycleLabelMachineFullSensor.Q	THEN //Czekanie na czujnik etykieciarki
										VIS.bBottleTransferRun					:=	TRUE;
									END_IF	
									
									IF P13_BottleTransfer.fbBottleTransfer.eRunningState>(1) THEN																																										
										iBottleTransferCase 				:=	2; 
										nCounterFormsToLoad					:=	1; //jedna formatka ma wyjechać
										//ctdCounterFormOnRobot.LOAD			:=	TRUE;
										nCounterForms						:=	0;
										eRobotPackageState[1].bBottleTransferedToLabeler := TRUE;	
										VIS.uiCounterGoodBottles			:=	VIS.uiCounterGoodBottles+1;	(*Liczenie dobrych opakowań*)(*Przeniesione*)
										VIS.udiCounterGlobal				:=	VIS.udiCounterGlobal+1;
										VIS.udiCounterShiftBottles		:=	VIS.udiCounterShiftBottles+1;	

										IF VIS.nBottleTransferPlaceOption	=	3 THEN
											bBottleTransferDoWeight					:= FALSE;
											VIS.bBottleTransferForceWeight			:= FALSE;
											udiBottleTransferWeightIntervalCount 	:= VIS.udiCounterGlobal;
										END_IF														
									END_IF									
								
							110: //Pobranie jednej i odłozenie na złe
									nCheckCountR4:=nCheckCountR4+1;
									VIS.nBottleTransferPickOption			:=	1; // 1 butelka
									VIS.nBottleTransferPlaceOption			:=	2; //odrzut zle butelki
									IF NOT tonCycleBadBottleConveyorFullSensor.Q THEN
										VIS.bBottleTransferRun				:=	TRUE;
									END_IF
									IF P13_BottleTransfer.fbBottleTransfer.eRunningState>1 THEN	
										iBottleTransferCase 				:= 2; 
										bAddGlobalCounter					:=	TRUE;
										bAddBadPackageReason				:=	TRUE;
										nCounterFormsToLoad					:=	1; // dwie formatki maja wyjechac
										//ctdCounterFormOnRobot.LOAD			:=	TRUE;
										nCounterForms						:=	0;										
										eRobotPackageState[1].bBottleTransferedToExit := TRUE;	
									END_IF
												
							120: //tylko wyjazd formatki jednej
										iBottleTransferCase 				:=	2; 
										nCounterFormsToLoad					:=	1; // dwie formatki maja wyjechac
										//ctdCounterFormOnRobot.LOAD			:=	TRUE;
										nCounterForms						:=	0;										
										eRobotPackageState[1].bBottleTransferedToExit := TRUE;								
											
							200: //Pobranie 2  i odłozenie dwóch butelki na dobre		
									nCheckCountR1:=nCheckCountR1+1;
									VIS.nBottleTransferPickOption			:=	2; // 1 butelka

									VIS.nBottleTransferPlaceOption			:=	1; //Dobre butelki 		
								
									IF 	bRobotPackageState1Rotate AND bRobotPackageState2Rotate THEN (* OBRÓT CHWYTAKA *)
										VIS.nBottleTransferPlaceOption		:=	4; 
									END_IF									
									
									IF tonCycleLabelMachineFullSensor.Q  THEN //Czekanie na czujnik etykieciarki
										VIS.bBottleTransferRun				:=	TRUE;
									END_IF										
									IF P13_BottleTransfer.fbBottleTransfer.eRunningState>1 THEN	
										iBottleTransferCase 				:=	2; 
										nCounterFormsToLoad					:=	2; //jedna formatka ma wyjechać
										//ctdCounterFormOnRobot.LOAD			:=	TRUE;
										nCounterForms						:=	0;										
										eRobotPackageState[1].bBottleTransferedToLabeler := TRUE;	
										eRobotPackageState[2].bBottleTransferedToLabeler := TRUE;
										(*Liczenie dobrych opakowań*)
										VIS.uiCounterGoodBottles			:=	VIS.uiCounterGoodBottles+2; //Przenieisone
										VIS.udiCounterGlobal				:=	VIS.udiCounterGlobal+2;
										VIS.udiCounterShiftBottles			:=	VIS.udiCounterShiftBottles+2;				
									END_IF									
							
							210: //Pobranie dwóch i odłozenie na złe
									nCheckCountR4:=nCheckCountR4+1;
									VIS.nBottleTransferPickOption			:=	2; // 2 butelka
									VIS.nBottleTransferPlaceOption			:=	2; //odrzut zle butelki
									IF NOT tonCycleBadBottleConveyorFullSensor.Q THEN
										VIS.bBottleTransferRun				:=	TRUE;
									END_IF
									IF P13_BottleTransfer.fbBottleTransfer.eRunningState>1 THEN	
										iBottleTransferCase 				:=	2; 
										nCounterFormsToLoad					:=	2; // dwie formatki maja wyjechac
										//ctdCounterFormOnRobot.LOAD			:=	TRUE;
										nCounterForms						:=	0;										
										bAddGlobalCounter					:=	TRUE;
										bAddBadPackageReason				:=	TRUE;
										bAddBadPackageReason2				:=	TRUE;
										eRobotPackageState[1].bBottleTransferedToExit := TRUE;	
										eRobotPackageState[2].bBottleTransferedToExit := TRUE;								
									END_IF
								
							220: //Wyjazd dwóch formatek bez odrzucania
									iBottleTransferCase 				:=	2; 
									nCounterFormsToLoad					:=	2; // dwie formatki maja wyjechac
									//ctdCounterFormOnRobot.LOAD			:=	TRUE;
									nCounterForms						:=	0;									
									eRobotPackageState[1].bBottleTransferedToExit := TRUE;	
									eRobotPackageState[2].bBottleTransferedToExit := TRUE;	
																		
					END_CASE

	2: //OTWORZENIE SZLABANU NA CZAS PRZEJAZDU FORMATEK
			iRobotPickCase := 0; //Nowe do stoppingu

			(*Spowalnianie transportera*)
			IF nCounterFormsToLoad = 1 AND eRobotPackageState[1].nCardNumber = ulFormTransportersScrewerSlowNumber AND eRobotPackageState[1].nCardNumber > 0 THEN
				bFormTransportersDispencerResetSpeed	:= TRUE;
				ulFormTransportersScrewerSlowNumber		:= 0;
			ELSIF  nCounterFormsToLoad = 2 AND 
					(
					(eRobotPackageState[1].nCardNumber = ulFormTransportersScrewerSlowNumber AND eRobotPackageState[1].nCardNumber >	0	)	OR
					(eRobotPackageState[2].nCardNumber = ulFormTransportersScrewerSlowNumber AND eRobotPackageState[2].nCardNumber >	0	) 
					)
			THEN
				bFormTransportersDispencerResetSpeed	:= TRUE;
				ulFormTransportersScrewerSlowNumber 	:=	0;
			END_IF
	
			//ctdCounterFormOnRobot.LOAD:=FALSE;
			IF NOT P01_Gates.fbGateRobot.bCycleDone	AND NOT fbIbBottleTransferFormAfterSensor.bOUT THEN
				VIS.bGateRobotEntranceRun				:= TRUE;
			END_IF
			//IF ctdCounterFormOnRobot.Q THEN
			IF nCounterForms >= nCounterFormsToLoad THEN				
				VIS.bGateRobotEntranceRun				:=	FALSE;
				bRobotStationDone						:=	TRUE;
				iBottleTransferCase						:=	3; 
			END_IF

	3: 
			IF (P13_BottleTransfer.fbBottleTransfer.bCycleDone OR NOT VIS.bBottleTransferRun) THEN
				VIS.bBottleTransferRun					:= FALSE;
				iBottleTransferCase						:=	4; 
				nCountTest3:=nCountTest3+1;
			END_IF
	4:		
			IF (((NOT (P00_PackML.fbPMLAuto.ePMLState = E_PMLState.ePMLState_STOPPING) OR P11_CapCorrectCheck.IbCapCorrectCheckAfterScrewerFormSensor) ) AND 				
					(P13_BottleTransfer.fbBottleTransfer.eState = E_Station.eReady AND NOT P13_BottleTransfer.fbBottleTransfer.bCycleDone)) 
				 OR NOT bBottleTransferEnable THEN
				iBottleTransferCase							:=	0; 
				nCountTest2:=nCountTest2+1;
			END_IF
END_CASE

//Zawsze dokańcza ruch place
VIS.bBottleTransferPlace :=TRUE;
END_ACTION

ACTION aP13_BottleTransferAfterDrag:
(*
Przeciaganie za robotem
tylko od czujników
*)

fbIbBottleTransferAfterDragAfterSensor		(bIN:=
											P00_PackML.fbPMLAuto.ePMLState = E_PMLState.ePMLState_EXECUTE AND P13_BottleTransferAfterDrag.IbBottleTransferAfterDragAfterSensor													
											,tFilterTimeOn:=T#0MS, tFilterTimeOff:=T#500MS);
fbIbBottleTransferAfterDragSecondFormSensor		(bIN:=
											P00_PackML.fbPMLAuto.ePMLState = E_PMLState.ePMLState_EXECUTE AND P13_BottleTransferAfterDrag.IbBottleTransferAfterDragSecondFormSensor													
											,tFilterTimeOn:=T#35MS, tFilterTimeOff:=T#35MS);
rtfbIbBottleTransferAfterDragSecondFormSensor (CLK:=fbIbBottleTransferAfterDragSecondFormSensor.bOUT,Q=>);
IF rtfbIbBottleTransferAfterDragSecondFormSensor.Q THEN
	rtfbIbBottleTransferAfterDragSecondFormSensorCounter := rtfbIbBottleTransferAfterDragSecondFormSensorCounter + 1;
END_IF
tonrtfbIbBottleTransferAfterDragSecondFormSensorCounter(IN:=	rtfbIbBottleTransferAfterDragSecondFormSensorCounter<2 AND 
																P13_BottleTransferAfterDrag.IbBottleTransferAfterDragFirstFormSensor AND
																P13_BottleTransferAfterDrag.IbBottleTransferAfterDragSecondFormSensor AND
																bFormTransportersAfterScrewerCmdStart
														,PT := T#10S);
IF tonrtfbIbBottleTransferAfterDragSecondFormSensorCounter.Q THEN
	rtfbIbBottleTransferAfterDragSecondFormSensorCounter := 2;
END_IF

tonBottleTransferAfterDrag (IN:= 
								(P00_PackML.fbPMLAuto.ePMLState = E_PMLState.ePMLState_EXECUTE) AND 
								NOT (P00_PackML.fbPMLAuto.ePMLState = E_PMLState.ePMLState_STOPPING) AND
								P13_BottleTransferAfterDrag.fbBottleTransferAfterDrag.eState = E_Station.eReady AND 

								P13_BottleTransferAfterDrag.IbBottleTransferAfterDragFirstFormSensor AND
								rtfbIbBottleTransferAfterDragSecondFormSensorCounter >=2 
								//P13_BottleTransferAfterDrag.IbBottleTransferAfterDragSecondFormSensor,	
							,PT:=T#0MS);
P01_PucksInserter.IbPucksInserterFormGateAfterSensor;// Czujnik za PI						
						
IF tonBottleTransferAfterDrag.Q AND 
	NOT P13_BottleTransferAfterDrag.fbBottleTransferAfterDrag.bCycleDone AND
	NOT fbIbBottleTransferAfterDragAfterSensor.bOUT
THEN
	VIS.bBottleTransferAfterDragRun	:= TRUE;
END_IF

IF P13_BottleTransferAfterDrag.fbBottleTransferAfterDrag.bCycleDone THEN
	VIS.bBottleTransferAfterDragRun	:= FALSE;
	rtfbIbBottleTransferAfterDragSecondFormSensorCounter:= 0;
END_IF
END_ACTION

ACTION aP14_BadBottleConveyor:

(*************TRANSPORTER ODRZUCONYCH BUTELEK****************)
(************Przeniesiono wyzej*****************************)

(*Załączany w programie robota jak jest dorzut butelki i kasowany po 30 sekundach*)
IF bBadBottleConveyorEnable THEN
	;
ELSE
	bBadBottleConveyorStart				:=	FALSE;
	bBadBottleConveyorStartTriggerDelay	:=	FALSE;
END_IF

//Opóznienie załączania transporeta
IF bBadBottleConveyorStartTriggerDelay AND P13_BottleTransfer.fbBottleTransfer.eRunningState = eRejected THEN
	bBadBottleConveyorStartTrigger			:= TRUE;
	bBadBottleConveyorStartTriggerDelay		:=FALSE;
END_IF

//Sterowanie transporterem odrzuconych butelek
rtBadBottleConvoyerStart	(CLK:=	bBadBottleConveyorStartTrigger);
tofBadBottleConveyorStart	(IN:=	rtBadBottleConvoyerStart.Q ,	PT:=T#10S);

IF rtBadBottleConvoyerStart.Q THEN //Uruchamianie na cykl
	bBadBottleConveyorStartTrigger		:=	FALSE;
END_IF
IF NOT tofBadBottleConveyorStart.Q  THEN
	bBadBottleConveyorStart				:=	FALSE;
	bBadBottleConveyorStartTrigger		:=	FALSE;
ELSE
	bBadBottleConveyorStart 			:=	TRUE;	
END_IF
END_ACTION

